MoveL RelTool (p1,30.000000,14.000000,15.535866,\Rx:=0.000000,\Ry:=-4.232438),vel1,zoneval,Extruder\WObj:=Workobject_1;
MoveL RelTool (p1,32.500000,14.000000,16.262071,\Rx:=0.000000,\Ry:=-3.021941),vel1,zoneval,Extruder\WObj:=Workobject_1;
MoveL RelTool (p1,35.000000,14.000000,16.795693,\Rx:=0.000000,\Ry:=-2.300490),vel1,zoneval,Extruder\WObj:=Workobject_1;
MoveL RelTool (p1,37.500000,14.000000,17.167850,\Rx:=0.000000,\Ry:=-1.460854),vel1,zoneval,Extruder\WObj:=Workobject_1;
MoveL RelTool (p1,40.000000,14.000000,17.403542,\Rx:=0.000000,\Ry:=-0.710383),vel1,zoneval,Extruder\WObj:=Workobject_1;
MoveL RelTool (p1,42.500000,14.000000,17.492358,\Rx:=0.000000,\Ry:=0.009614),vel1,zoneval,Extruder\WObj:=Workobject_1;
MoveL RelTool (p1,45.000000,14.000000,17.445886,\Rx:=0.000000,\Ry:=0.497915),vel1,zoneval,Extruder\WObj:=Workobject_1;
MoveL RelTool (p1,47.500000,14.000000,17.268613,\Rx:=0.000000,\Ry:=1.477311),vel1,zoneval,Extruder\WObj:=Workobject_1;
MoveL RelTool (p1,50.000000,14.000000,16.934162,\Rx:=0.000000,\Ry:=1.958454),vel1,zoneval,Extruder\WObj:=Workobject_1;
MoveL RelTool (p1,52.500000,14.000000,16.462457,\Rx:=0.000000,\Ry:=3.004009),vel1,zoneval,Extruder\WObj:=Workobject_1;
MoveL RelTool (p1,55.000000,14.000000,15.799199,\Rx:=0.000000,\Ry:=3.621934),vel1,zoneval,Extruder\WObj:=Workobject_1;
MoveL RelTool (p1,57.500000,14.000000,14.938044,\Rx:=0.000000,\Ry:=4.715755),vel1,zoneval,Extruder\WObj:=Workobject_1;
MoveL RelTool (p1,60.000000,14.000000,13.810971,\Rx:=0.000000,\Ry:=6.022619),vel1,zoneval,Extruder\WObj:=Workobject_1;
MoveL RelTool (p1,62.500000,14.000000,12.303856,\Rx:=0.000000,\Ry:=8.132481),vel1,zoneval,Extruder\WObj:=Workobject_1;
MoveL RelTool (p1,65.000000,14.000000,10.061417,\Rx:=0.000000,\Ry:=11.488801),vel1,zoneval,Extruder\WObj:=Workobject_1;
MoveL RelTool (p1,67.500000,14.000000,7.780757,\Rx:=0.000000,\Ry:=3.821551),vel1,zoneval,Extruder\WObj:=Workobject_1;
MoveL RelTool (p1,70.000000,14.000000,7.500000,\Rx:=0.000000,\Ry:=-0.000000),vel1,zoneval,Extruder\WObj:=Workobject_1;
MoveL RelTool (p1,72.500000,14.000000,7.500000,\Rx:=0.000000,\Ry:=-0.000000),vel1,zoneval,Extruder\WObj:=Workobject_1;
MoveL RelTool (p1,75.000000,14.000000,7.500000,\Rx:=0.000000,\Ry:=-0.000000),vel1,zoneval,Extruder\WObj:=Workobject_1;
MoveL RelTool (p1,77.500000,14.000000,7.500000,\Rx:=0.000000,\Ry:=-0.000000),vel1,zoneval,Extruder\WObj:=Workobject_1;
MoveL RelTool (p1,80.000000,14.000000,7.500000,\Rx:=0.000000,\Ry:=-0.000000),vel1,zoneval,Extruder\WObj:=Workobject_1;
MoveL RelTool (p1,82.500000,14.000000,7.500000,\Rx:=0.000000,\Ry:=-0.000000),vel1,zoneval,Extruder\WObj:=Workobject_1;
MoveL RelTool (p1,80.500000,14.500000,7.500000,\Rx:=0.000000,\Ry:=0.000000),vel1,zoneval,Extruder\WObj:=Workobject_1;
MoveL RelTool (p1,78.000000,14.500000,7.500000,\Rx:=0.000000,\Ry:=0.000000),vel1,zoneval,Extruder\WObj:=Workobject_1;
MoveL RelTool (p1,75.500000,14.500000,7.500000,\Rx:=0.000000,\Ry:=0.000000),vel1,zoneval,Extruder\WObj:=Workobject_1;
MoveL RelTool (p1,73.000000,14.500000,7.500000,\Rx:=0.000000,\Ry:=0.000000),vel1,zoneval,Extruder\WObj:=Workobject_1;
MoveL RelTool (p1,70.500000,14.500000,7.500000,\Rx:=0.000000,\Ry:=0.000000),vel1,zoneval,Extruder\WObj:=Workobject_1;
MoveL RelTool (p1,68.000000,14.500000,7.626010,\Rx:=0.000000,\Ry:=3.821551),vel1,zoneval,Extruder\WObj:=Workobject_1;
MoveL RelTool (p1,65.500000,14.500000,9.428317,\Rx:=0.000000,\Ry:=11.485360),vel1,zoneval,Extruder\WObj:=Workobject_1;
MoveL RelTool (p1,63.000000,14.500000,11.932892,\Rx:=0.000000,\Ry:=8.132481),vel1,zoneval,Extruder\WObj:=Workobject_1;
MoveL RelTool (p1,60.500000,14.500000,13.554932,\Rx:=0.000000,\Ry:=6.053141),vel1,zoneval,Extruder\WObj:=Workobject_1;
MoveL RelTool (p1,58.000000,14.500000,14.744603,\Rx:=0.000000,\Ry:=4.711369),vel1,zoneval,Extruder\WObj:=Workobject_1;
MoveL RelTool (p1,55.500000,14.500000,15.652731,\Rx:=0.000000,\Ry:=3.666878),vel1,zoneval,Extruder\WObj:=Workobject_1;
MoveL RelTool (p1,53.000000,14.500000,16.342269,\Rx:=0.000000,\Ry:=3.014175),vel1,zoneval,Extruder\WObj:=Workobject_1;
MoveL RelTool (p1,50.500000,14.500000,16.857119,\Rx:=0.000000,\Ry:=1.968139),vel1,zoneval,Extruder\WObj:=Workobject_1;
MoveL RelTool (p1,48.000000,14.500000,17.210020,\Rx:=0.000000,\Ry:=1.477311),vel1,zoneval,Extruder\WObj:=Workobject_1;
MoveL RelTool (p1,45.500000,14.500000,17.426141,\Rx:=0.000000,\Ry:=0.497915),vel1,zoneval,Extruder\WObj:=Workobject_1;
MoveL RelTool (p1,43.000000,14.500000,17.491866,\Rx:=0.000000,\Ry:=0.009614),vel1,zoneval,Extruder\WObj:=Workobject_1;
MoveL RelTool (p1,40.500000,14.500000,17.432366,\Rx:=0.000000,\Ry:=-0.740871),vel1,zoneval,Extruder\WObj:=Workobject_1;
MoveL RelTool (p1,38.000000,14.500000,17.226111,\Rx:=0.000000,\Ry:=-1.460854),vel1,zoneval,Extruder\WObj:=Workobject_1;
MoveL RelTool (p1,35.500000,14.500000,16.886724,\Rx:=0.000000,\Ry:=-2.257683),vel1,zoneval,Extruder\WObj:=Workobject_1;
MoveL RelTool (p1,33.000000,14.500000,16.382907,\Rx:=0.000000,\Ry:=-3.021941),vel1,zoneval,Extruder\WObj:=Workobject_1;
MoveL RelTool (p1,30.500000,14.500000,15.708835,\Rx:=0.000000,\Ry:=-4.213102),vel1,zoneval,Extruder\WObj:=Workobject_1;
MoveL RelTool (p1,28.000000,14.500000,14.810880,\Rx:=0.000000,\Ry:=-5.088446),vel1,zoneval,Extruder\WObj:=Workobject_1;
MoveL RelTool (p1,25.500000,14.500000,13.645137,\Rx:=0.000000,\Ry:=-6.516459),vel1,zoneval,Extruder\WObj:=Workobject_1;
MoveL RelTool (p1,23.000000,14.500000,12.058948,\Rx:=0.000000,\Ry:=-8.297239),vel1,zoneval,Extruder\WObj:=Workobject_1;
MoveL RelTool (p1,20.500000,14.500000,9.662581,\Rx:=0.000000,\Ry:=-11.719870),vel1,zoneval,Extruder\WObj:=Workobject_1;
MoveL RelTool (p1,18.000000,14.500000,7.667393,\Rx:=0.000000,\Ry:=-2.952187),vel1,zoneval,Extruder\WObj:=Workobject_1;
MoveL RelTool (p1,15.500000,14.500000,7.500000,\Rx:=0.000000,\Ry:=0.000000),vel1,zoneval,Extruder\WObj:=Workobject_1;
MoveL RelTool (p1,13.000000,14.500000,7.500000,\Rx:=0.000000,\Ry:=0.000000),vel1,zoneval,Extruder\WObj:=Workobject_1;
MoveL RelTool (p1,10.500000,14.500000,7.500000,\Rx:=0.000000,\Ry:=0.000000),vel1,zoneval,Extruder\WObj:=Workobject_1;
MoveL RelTool (p1,8.000000,14.500000,7.500000,\Rx:=0.000000,\Ry:=0.000000),vel1,zoneval,Extruder\WObj:=Workobject_1;
MoveL RelTool (p1,5.500000,14.500000,7.500000,\Rx:=0.000000,\Ry:=0.000000),vel1,zoneval,Extruder\WObj:=Workobject_1;
MoveL RelTool (p1,3.000000,14.500000,7.500000,\Rx:=0.000000,\Ry:=0.000000),vel1,zoneval,Extruder\WObj:=Workobject_1;
MoveL RelTool (p1,5.000000,15.000000,7.500000,\Rx:=0.000000,\Ry:=-0.000000),vel1,zoneval,Extruder\WObj:=Workobject_1;
MoveL RelTool (p1,7.500000,15.000000,7.500000,\Rx:=0.000000,\Ry:=-0.000000),vel1,zoneval,Extruder\WObj:=Workobject_1;
MoveL RelTool (p1,10.000000,15.000000,7.500000,\Rx:=0.000000,\Ry:=-0.000000),vel1,zoneval,Extruder\WObj:=Workobject_1;
MoveL RelTool (p1,12.500000,15.000000,7.500000,\Rx:=0.000000,\Ry:=-0.000000),vel1,zoneval,Extruder\WObj:=Workobject_1;
MoveL RelTool (p1,15.000000,15.000000,7.500000,\Rx:=0.000000,\Ry:=-0.000000),vel1,zoneval,Extruder\WObj:=Workobject_1;
MoveL RelTool (p1,17.500000,15.000000,7.549338,\Rx:=0.000000,\Ry:=-2.952187),vel1,zoneval,Extruder\WObj:=Workobject_1;
MoveL RelTool (p1,20.000000,15.000000,9.005299,\Rx:=0.000000,\Ry:=-11.718071),vel1,zoneval,Extruder\WObj:=Workobject_1;
MoveL RelTool (p1,22.500000,15.000000,11.677302,\Rx:=0.000000,\Ry:=-8.297239),vel1,zoneval,Extruder\WObj:=Workobject_1;
MoveL RelTool (p1,25.000000,15.000000,13.364411,\Rx:=0.000000,\Ry:=-6.507557),vel1,zoneval,Extruder\WObj:=Workobject_1;
MoveL RelTool (p1,27.500000,15.000000,14.600606,\Rx:=0.000000,\Ry:=-5.061360),vel1,zoneval,Extruder\WObj:=Workobject_1;
MoveL RelTool (p1,30.000000,15.000000,15.538278,\Rx:=0.000000,\Ry:=-4.191749),vel1,zoneval,Extruder\WObj:=Workobject_1;
MoveL RelTool (p1,32.500000,15.000000,16.261840,\Rx:=0.000000,\Ry:=-3.021941),vel1,zoneval,Extruder\WObj:=Workobject_1;
MoveL RelTool (p1,35.000000,15.000000,16.798556,\Rx:=0.000000,\Ry:=-2.214824),vel1,zoneval,Extruder\WObj:=Workobject_1;
MoveL RelTool (p1,37.500000,15.000000,17.169131,\Rx:=0.000000,\Ry:=-1.460854),vel1,zoneval,Extruder\WObj:=Workobject_1;
MoveL RelTool (p1,40.000000,15.000000,17.402936,\Rx:=0.000000,\Ry:=-0.761113),vel1,zoneval,Extruder\WObj:=Workobject_1;
MoveL RelTool (p1,42.500000,15.000000,17.492129,\Rx:=0.000000,\Ry:=0.009614),vel1,zoneval,Extruder\WObj:=Workobject_1;
MoveL RelTool (p1,45.000000,15.000000,17.445523,\Rx:=0.000000,\Ry:=0.497915),vel1,zoneval,Extruder\WObj:=Workobject_1;
MoveL RelTool (p1,47.500000,15.000000,17.267978,\Rx:=0.000000,\Ry:=1.477311),vel1,zoneval,Extruder\WObj:=Workobject_1;
MoveL RelTool (p1,50.000000,15.000000,16.935897,\Rx:=0.000000,\Ry:=1.976483),vel1,zoneval,Extruder\WObj:=Workobject_1;
MoveL RelTool (p1,52.500000,15.000000,16.462915,\Rx:=0.000000,\Ry:=3.014175),vel1,zoneval,Extruder\WObj:=Workobject_1;
MoveL RelTool (p1,55.000000,15.000000,15.802495,\Rx:=0.000000,\Ry:=3.711728),vel1,zoneval,Extruder\WObj:=Workobject_1;
MoveL RelTool (p1,57.500000,15.000000,14.939061,\Rx:=0.000000,\Ry:=4.706981),vel1,zoneval,Extruder\WObj:=Workobject_1;
MoveL RelTool (p1,60.000000,15.000000,13.813687,\Rx:=0.000000,\Ry:=6.083587),vel1,zoneval,Extruder\WObj:=Workobject_1;
MoveL RelTool (p1,62.500000,15.000000,12.304491,\Rx:=0.000000,\Ry:=8.132481),vel1,zoneval,Extruder\WObj:=Workobject_1;
MoveL RelTool (p1,65.000000,15.000000,10.060714,\Rx:=0.000000,\Ry:=11.481917),vel1,zoneval,Extruder\WObj:=Workobject_1;
MoveL RelTool (p1,67.500000,15.000000,7.780757,\Rx:=0.000000,\Ry:=3.821551),vel1,zoneval,Extruder\WObj:=Workobject_1;
MoveL RelTool (p1,70.000000,15.000000,7.500000,\Rx:=0.000000,\Ry:=-0.000000),vel1,zoneval,Extruder\WObj:=Workobject_1;
MoveL RelTool (p1,72.500000,15.000000,7.500000,\Rx:=0.000000,\Ry:=-0.000000),vel1,zoneval,Extruder\WObj:=Workobject_1;
MoveL RelTool (p1,75.000000,15.000000,7.500000,\Rx:=0.000000,\Ry:=-0.000000),vel1,zoneval,Extruder\WObj:=Workobject_1;
MoveL RelTool (p1,77.500000,15.000000,7.500000,\Rx:=0.000000,\Ry:=-0.000000),vel1,zoneval,Extruder\WObj:=Workobject_1;
MoveL RelTool (p1,80.000000,15.000000,7.500000,\Rx:=0.000000,\Ry:=-0.000000),vel1,zoneval,Extruder\WObj:=Workobject_1;
MoveL RelTool (p1,82.500000,15.000000,7.500000,\Rx:=0.000000,\Ry:=-0.000000),vel1,zoneval,Extruder\WObj:=Workobject_1;
MoveL RelTool (p1,80.500000,15.500000,7.500000,\Rx:=0.000000,\Ry:=0.000000),vel1,zoneval,Extruder\WObj:=Workobject_1;
MoveL RelTool (p1,78.000000,15.500000,7.500000,\Rx:=0.000000,\Ry:=0.000000),vel1,zoneval,Extruder\WObj:=Workobject_1;
MoveL RelTool (p1,75.500000,15.500000,7.500000,\Rx:=0.000000,\Ry:=0.000000),vel1,zoneval,Extruder\WObj:=Workobject_1;
MoveL RelTool (p1,73.000000,15.500000,7.500000,\Rx:=0.000000,\Ry:=0.000000),vel1,zoneval,Extruder\WObj:=Workobject_1;
MoveL RelTool (p1,70.500000,15.500000,7.500000,\Rx:=0.000000,\Ry:=0.000000),vel1,zoneval,Extruder\WObj:=Workobject_1;
MoveL RelTool (p1,68.000000,15.500000,7.626010,\Rx:=0.000000,\Ry:=3.821551),vel1,zoneval,Extruder\WObj:=Workobject_1;
MoveL RelTool (p1,65.500000,15.500000,9.428317,\Rx:=0.000000,\Ry:=11.478472),vel1,zoneval,Extruder\WObj:=Workobject_1;
MoveL RelTool (p1,63.000000,15.500000,11.933528,\Rx:=0.000000,\Ry:=8.132481),vel1,zoneval,Extruder\WObj:=Workobject_1;
MoveL RelTool (p1,60.500000,15.500000,13.554619,\Rx:=0.000000,\Ry:=6.113959),vel1,zoneval,Extruder\WObj:=Workobject_1;
MoveL RelTool (p1,58.000000,15.500000,14.746017,\Rx:=0.000000,\Ry:=4.702592),vel1,zoneval,Extruder\WObj:=Workobject_1;
MoveL RelTool (p1,55.500000,15.500000,15.652192,\Rx:=0.000000,\Ry:=3.756483),vel1,zoneval,Extruder\WObj:=Workobject_1;
MoveL RelTool (p1,53.000000,15.500000,16.342305,\Rx:=0.000000,\Ry:=3.014175),vel1,zoneval,Extruder\WObj:=Workobject_1;
MoveL RelTool (p1,50.500000,15.500000,16.858518,\Rx:=0.000000,\Ry:=1.976483),vel1,zoneval,Extruder\WObj:=Workobject_1;
MoveL RelTool (p1,48.000000,15.500000,17.209385,\Rx:=0.000000,\Ry:=1.477311),vel1,zoneval,Extruder\WObj:=Workobject_1;
MoveL RelTool (p1,45.500000,15.500000,17.425779,\Rx:=0.000000,\Ry:=0.497915),vel1,zoneval,Extruder\WObj:=Workobject_1;
MoveL RelTool (p1,43.000000,15.500000,17.491637,\Rx:=0.000000,\Ry:=0.009614),vel1,zoneval,Extruder\WObj:=Workobject_1;
MoveL RelTool (p1,40.500000,15.500000,17.433003,\Rx:=0.000000,\Ry:=-0.772436),vel1,zoneval,Extruder\WObj:=Workobject_1;
MoveL RelTool (p1,38.000000,15.500000,17.227393,\Rx:=0.000000,\Ry:=-1.460854),vel1,zoneval,Extruder\WObj:=Workobject_1;
MoveL RelTool (p1,35.500000,15.500000,16.886115,\Rx:=0.000000,\Ry:=-2.171914),vel1,zoneval,Extruder\WObj:=Workobject_1;
MoveL RelTool (p1,33.000000,15.500000,16.382676,\Rx:=0.000000,\Ry:=-3.021941),vel1,zoneval,Extruder\WObj:=Workobject_1;
MoveL RelTool (p1,30.500000,15.500000,15.708951,\Rx:=0.000000,\Ry:=-4.160740),vel1,zoneval,Extruder\WObj:=Workobject_1;
MoveL RelTool (p1,28.000000,15.500000,14.810202,\Rx:=0.000000,\Ry:=-5.034225),vel1,zoneval,Extruder\WObj:=Workobject_1;
MoveL RelTool (p1,25.500000,15.500000,13.644491,\Rx:=0.000000,\Ry:=-6.498647),vel1,zoneval,Extruder\WObj:=Workobject_1;
MoveL RelTool (p1,23.000000,15.500000,12.058489,\Rx:=0.000000,\Ry:=-8.297239),vel1,zoneval,Extruder\WObj:=Workobject_1;
MoveL RelTool (p1,20.500000,15.500000,9.662195,\Rx:=0.000000,\Ry:=-11.716271),vel1,zoneval,Extruder\WObj:=Workobject_1;
MoveL RelTool (p1,18.000000,15.500000,7.667393,\Rx:=0.000000,\Ry:=-2.952187),vel1,zoneval,Extruder\WObj:=Workobject_1;
MoveL RelTool (p1,15.500000,15.500000,7.500000,\Rx:=0.000000,\Ry:=0.000000),vel1,zoneval,Extruder\WObj:=Workobject_1;
MoveL RelTool (p1,13.000000,15.500000,7.500000,\Rx:=0.000000,\Ry:=0.000000),vel1,zoneval,Extruder\WObj:=Workobject_1;
MoveL RelTool (p1,10.500000,15.500000,7.500000,\Rx:=0.000000,\Ry:=0.000000),vel1,zoneval,Extruder\WObj:=Workobject_1;
MoveL RelTool (p1,8.000000,15.500000,7.500000,\Rx:=0.000000,\Ry:=0.000000),vel1,zoneval,Extruder\WObj:=Workobject_1;
MoveL RelTool (p1,5.500000,15.500000,7.500000,\Rx:=0.000000,\Ry:=0.000000),vel1,zoneval,Extruder\WObj:=Workobject_1;
MoveL RelTool (p1,3.000000,15.500000,7.500000,\Rx:=0.000000,\Ry:=0.000000),vel1,zoneval,Extruder\WObj:=Workobject_1;
MoveL RelTool (p1,5.000000,16.000000,7.500000,\Rx:=0.000000,\Ry:=-0.000000),vel1,zoneval,Extruder\WObj:=Workobject_1;
MoveL RelTool (p1,7.500000,16.000000,7.500000,\Rx:=0.000000,\Ry:=-0.000000),vel1,zoneval,Extruder\WObj:=Workobject_1;
MoveL RelTool (p1,10.000000,16.000000,7.500000,\Rx:=0.000000,\Ry:=-0.000000),vel1,zoneval,Extruder\WObj:=Workobject_1;
MoveL RelTool (p1,12.500000,16.000000,7.500000,\Rx:=0.000000,\Ry:=-0.000000),vel1,zoneval,Extruder\WObj:=Workobject_1;
MoveL RelTool (p1,15.000000,16.000000,7.500000,\Rx:=0.000000,\Ry:=-0.000000),vel1,zoneval,Extruder\WObj:=Workobject_1;
MoveL RelTool (p1,17.500000,16.000000,7.549338,\Rx:=0.000000,\Ry:=-2.952187),vel1,zoneval,Extruder\WObj:=Workobject_1;
MoveL RelTool (p1,20.000000,16.000000,9.005299,\Rx:=0.000000,\Ry:=-11.714470),vel1,zoneval,Extruder\WObj:=Workobject_1;
MoveL RelTool (p1,22.500000,16.000000,11.676843,\Rx:=0.000000,\Ry:=-8.297239),vel1,zoneval,Extruder\WObj:=Workobject_1;
MoveL RelTool (p1,25.000000,16.000000,13.364684,\Rx:=0.000000,\Ry:=-6.489730),vel1,zoneval,Extruder\WObj:=Workobject_1;
MoveL RelTool (p1,27.500000,16.000000,14.602432,\Rx:=0.000000,\Ry:=-5.007042),vel1,zoneval,Extruder\WObj:=Workobject_1;
MoveL RelTool (p1,30.000000,16.000000,15.540690,\Rx:=0.000000,\Ry:=-4.129681),vel1,zoneval,Extruder\WObj:=Workobject_1;
MoveL RelTool (p1,32.500000,16.000000,16.261609,\Rx:=0.000000,\Ry:=-3.021941),vel1,zoneval,Extruder\WObj:=Workobject_1;
MoveL RelTool (p1,35.000000,16.000000,16.801419,\Rx:=0.000000,\Ry:=-2.128954),vel1,zoneval,Extruder\WObj:=Workobject_1;
MoveL RelTool (p1,37.500000,16.000000,17.170413,\Rx:=0.000000,\Ry:=-1.460854),vel1,zoneval,Extruder\WObj:=Workobject_1;
MoveL RelTool (p1,40.000000,16.000000,17.402329,\Rx:=0.000000,\Ry:=-0.783758),vel1,zoneval,Extruder\WObj:=Workobject_1;
MoveL RelTool (p1,42.500000,16.000000,17.491899,\Rx:=0.000000,\Ry:=0.009614),vel1,zoneval,Extruder\WObj:=Workobject_1;
MoveL RelTool (p1,45.000000,16.000000,17.445161,\Rx:=0.000000,\Ry:=0.497915),vel1,zoneval,Extruder\WObj:=Workobject_1;
MoveL RelTool (p1,47.500000,16.000000,17.267343,\Rx:=0.000000,\Ry:=1.477311),vel1,zoneval,Extruder\WObj:=Workobject_1;
MoveL RelTool (p1,50.000000,16.000000,16.937631,\Rx:=0.000000,\Ry:=1.976483),vel1,zoneval,Extruder\WObj:=Workobject_1;
MoveL RelTool (p1,52.500000,16.000000,16.462951,\Rx:=0.000000,\Ry:=3.014175),vel1,zoneval,Extruder\WObj:=Workobject_1;
MoveL RelTool (p1,55.000000,16.000000,15.805792,\Rx:=0.000000,\Ry:=3.801143),vel1,zoneval,Extruder\WObj:=Workobject_1;
MoveL RelTool (p1,57.500000,16.000000,14.940078,\Rx:=0.000000,\Ry:=4.700199),vel1,zoneval,Extruder\WObj:=Workobject_1;
MoveL RelTool (p1,60.000000,16.000000,13.816402,\Rx:=0.000000,\Ry:=6.144255),vel1,zoneval,Extruder\WObj:=Workobject_1;
MoveL RelTool (p1,62.500000,16.000000,12.305126,\Rx:=0.000000,\Ry:=8.132481),vel1,zoneval,Extruder\WObj:=Workobject_1;
MoveL RelTool (p1,65.000000,16.000000,10.060011,\Rx:=0.000000,\Ry:=11.475024),vel1,zoneval,Extruder\WObj:=Workobject_1;
MoveL RelTool (p1,67.500000,16.000000,7.780757,\Rx:=0.000000,\Ry:=3.821551),vel1,zoneval,Extruder\WObj:=Workobject_1;
MoveL RelTool (p1,70.000000,16.000000,7.500000,\Rx:=0.000000,\Ry:=-0.000000),vel1,zoneval,Extruder\WObj:=Workobject_1;
MoveL RelTool (p1,72.500000,16.000000,7.500000,\Rx:=0.000000,\Ry:=-0.000000),vel1,zoneval,Extruder\WObj:=Workobject_1;
MoveL RelTool (p1,75.000000,16.000000,7.500000,\Rx:=0.000000,\Ry:=-0.000000),vel1,zoneval,Extruder\WObj:=Workobject_1;
MoveL RelTool (p1,77.500000,16.000000,7.500000,\Rx:=0.000000,\Ry:=-0.000000),vel1,zoneval,Extruder\WObj:=Workobject_1;
MoveL RelTool (p1,80.000000,16.000000,7.500000,\Rx:=0.000000,\Ry:=-0.000000),vel1,zoneval,Extruder\WObj:=Workobject_1;
MoveL RelTool (p1,82.500000,16.000000,7.500000,\Rx:=0.000000,\Ry:=-0.000000),vel1,zoneval,Extruder\WObj:=Workobject_1;




MoveL RelTool (p1,82.500000,16.000000,70.00000,\Rx:=0.000000,\Ry:=-0.000000),vel1,zoneval,Extruder\WObj:=Workobject_1;


MoveL RelTool (p1,3.000000,3.000000,70.000000,\Rx:=0.000000,\Ry:=0.000000),vel1,z0,Extruder\WObj:=Workobject_1;

MoveL RelTool (p1,3.000000,3.000000,8.000000,\Rx:=0.000000,\Ry:=0.000000),vel1,z0,Extruder\WObj:=Workobject_1;
MoveL RelTool (p1,16.889791,3.000000,8.000000,\Rx:=0.000000,\Ry:=0.000000),vel1,z0,Extruder\WObj:=Workobject_1;
MoveL RelTool (p1,17.452093,3.000000,8.045464,\Rx:=0.000000,\Ry:=0.000000),vel1,z0,Extruder\WObj:=Workobject_1;
MoveL RelTool (p1,17.999786,3.000000,8.180676,\Rx:=0.000000,\Ry:=0.000000),vel1,z0,Extruder\WObj:=Workobject_1;
MoveL RelTool (p1,18.518642,3.000000,8.402122,\Rx:=0.000000,\Ry:=0.000000),vel1,z0,Extruder\WObj:=Workobject_1;
MoveL RelTool (p1,18.995180,3.000000,8.704050,\Rx:=0.000000,\Ry:=0.000000),vel1,z0,Extruder\WObj:=Workobject_1;
MoveL RelTool (p1,19.417023,3.000000,9.078616,\Rx:=0.000000,\Ry:=0.000000),vel1,z0,Extruder\WObj:=Workobject_1;
MoveL RelTool (p1,19.773207,3.000000,9.516088,\Rx:=0.000000,\Ry:=0.000000),vel1,z0,Extruder\WObj:=Workobject_1;
MoveL RelTool (p1,20.250246,3.000000,10.153003,\Rx:=0.000000,\Ry:=0.000000),vel1,z0,Extruder\WObj:=Workobject_1;
MoveL RelTool (p1,21.342972,3.000000,11.327476,\Rx:=0.000000,\Ry:=0.000000),vel1,z0,Extruder\WObj:=Workobject_1;
MoveL RelTool (p1,22.725681,3.000000,12.487259,\Rx:=0.000000,\Ry:=0.000000),vel1,z0,Extruder\WObj:=Workobject_1;
MoveL RelTool (p1,24.403374,3.000000,13.604031,\Rx:=0.000000,\Ry:=0.000000),vel1,z0,Extruder\WObj:=Workobject_1;
MoveL RelTool (p1,26.408426,3.000000,14.665359,\Rx:=0.000000,\Ry:=0.000000),vel1,z0,Extruder\WObj:=Workobject_1;
MoveL RelTool (p1,28.691647,3.000000,15.620553,\Rx:=0.000000,\Ry:=0.000000),vel1,z0,Extruder\WObj:=Workobject_1;
MoveL RelTool (p1,31.195286,3.000000,16.437975,\Rx:=0.000000,\Ry:=0.000000),vel1,z0,Extruder\WObj:=Workobject_1;
MoveL RelTool (p1,33.926628,3.000000,17.106159,\Rx:=0.000000,\Ry:=0.000000),vel1,z0,Extruder\WObj:=Workobject_1;
MoveL RelTool (p1,36.846878,3.000000,17.599693,\Rx:=0.000000,\Ry:=0.000000),vel1,z0,Extruder\WObj:=Workobject_1;
MoveL RelTool (p1,39.856747,3.000000,17.899025,\Rx:=0.000000,\Ry:=0.000000),vel1,z0,Extruder\WObj:=Workobject_1;
MoveL RelTool (p1,42.916187,3.000000,18.000000,\Rx:=0.000000,\Ry:=0.000000),vel1,z0,Extruder\WObj:=Workobject_1;
MoveL RelTool (p1,45.700897,3.000000,17.916361,\Rx:=0.000000,\Ry:=0.000000),vel1,z0,Extruder\WObj:=Workobject_1;
MoveL RelTool (p1,48.678219,3.000000,17.639635,\Rx:=0.000000,\Ry:=0.000000),vel1,z0,Extruder\WObj:=Workobject_1;
MoveL RelTool (p1,51.519215,3.000000,17.183882,\Rx:=0.000000,\Ry:=0.000000),vel1,z0,Extruder\WObj:=Workobject_1;
MoveL RelTool (p1,54.218540,3.000000,16.554611,\Rx:=0.000000,\Ry:=0.000000),vel1,z0,Extruder\WObj:=Workobject_1;
MoveL RelTool (p1,56.711525,3.000000,15.776219,\Rx:=0.000000,\Ry:=0.000000),vel1,z0,Extruder\WObj:=Workobject_1;
MoveL RelTool (p1,58.923611,3.000000,14.894774,\Rx:=0.000000,\Ry:=0.000000),vel1,z0,Extruder\WObj:=Workobject_1;
MoveL RelTool (p1,60.880539,3.000000,13.919682,\Rx:=0.000000,\Ry:=0.000000),vel1,z0,Extruder\WObj:=Workobject_1;
MoveL RelTool (p1,62.570816,3.000000,12.872232,\Rx:=0.000000,\Ry:=0.000000),vel1,z0,Extruder\WObj:=Workobject_1;
MoveL RelTool (p1,63.995117,3.000000,11.774377,\Rx:=0.000000,\Ry:=0.000000),vel1,z0,Extruder\WObj:=Workobject_1;
MoveL RelTool (p1,65.148392,3.000000,10.656720,\Rx:=0.000000,\Ry:=0.000000),vel1,z0,Extruder\WObj:=Workobject_1;
MoveL RelTool (p1,66.059166,3.000000,9.516088,\Rx:=0.000000,\Ry:=0.000000),vel1,z0,Extruder\WObj:=Workobject_1;
MoveL RelTool (p1,66.415344,3.000000,9.078616,\Rx:=0.000000,\Ry:=0.000000),vel1,z0,Extruder\WObj:=Workobject_1;
MoveL RelTool (p1,66.837189,3.000000,8.704050,\Rx:=0.000000,\Ry:=0.000000),vel1,z0,Extruder\WObj:=Workobject_1;
MoveL RelTool (p1,67.313728,3.000000,8.402122,\Rx:=0.000000,\Ry:=0.000000),vel1,z0,Extruder\WObj:=Workobject_1;
MoveL RelTool (p1,67.832588,3.000000,8.180676,\Rx:=0.000000,\Ry:=0.000000),vel1,z0,Extruder\WObj:=Workobject_1;
MoveL RelTool (p1,68.380280,3.000000,8.045464,\Rx:=0.000000,\Ry:=0.000000),vel1,z0,Extruder\WObj:=Workobject_1;
MoveL RelTool (p1,68.942581,3.000000,8.000000,\Rx:=0.000000,\Ry:=0.000000),vel1,z0,Extruder\WObj:=Workobject_1;
MoveL RelTool (p1,82.832375,3.000000,8.000000,\Rx:=0.000000,\Ry:=0.000000),vel1,z0,Extruder\WObj:=Workobject_1;
MoveL RelTool (p1,82.832375,16.000000,8.000000,\Rx:=0.000000,\Ry:=0.000000),vel1,z0,Extruder\WObj:=Workobject_1;
MoveL RelTool (p1,68.942581,16.000000,8.000000,\Rx:=0.000000,\Ry:=0.000000),vel1,z0,Extruder\WObj:=Workobject_1;
MoveL RelTool (p1,68.380280,16.000000,8.045464,\Rx:=0.000000,\Ry:=0.000000),vel1,z0,Extruder\WObj:=Workobject_1;
MoveL RelTool (p1,67.832588,16.000000,8.180676,\Rx:=0.000000,\Ry:=0.000000),vel1,z0,Extruder\WObj:=Workobject_1;
MoveL RelTool (p1,67.313728,16.000000,8.402122,\Rx:=0.000000,\Ry:=0.000000),vel1,z0,Extruder\WObj:=Workobject_1;
MoveL RelTool (p1,66.837189,16.000000,8.704050,\Rx:=0.000000,\Ry:=0.000000),vel1,z0,Extruder\WObj:=Workobject_1;
MoveL RelTool (p1,66.415344,16.000000,9.078616,\Rx:=0.000000,\Ry:=0.000000),vel1,z0,Extruder\WObj:=Workobject_1;
MoveL RelTool (p1,66.059166,16.000000,9.516088,\Rx:=0.000000,\Ry:=0.000000),vel1,z0,Extruder\WObj:=Workobject_1;
MoveL RelTool (p1,65.564453,16.000000,10.174875,\Rx:=0.000000,\Ry:=0.000000),vel1,z0,Extruder\WObj:=Workobject_1;
MoveL RelTool (p1,65.143768,16.000000,10.652657,\Rx:=0.000000,\Ry:=0.000000),vel1,z0,Extruder\WObj:=Workobject_1;
MoveL RelTool (p1,64.991638,16.000000,10.825450,\Rx:=0.000000,\Ry:=0.000000),vel1,z0,Extruder\WObj:=Workobject_1;
MoveL RelTool (p1,64.322777,16.000000,11.482923,\Rx:=0.000000,\Ry:=0.000000),vel1,z0,Extruder\WObj:=Workobject_1;
MoveL RelTool (p1,63.989872,16.000000,11.768258,\Rx:=0.000000,\Ry:=0.000000),vel1,z0,Extruder\WObj:=Workobject_1;
MoveL RelTool (p1,63.561058,16.000000,12.135797,\Rx:=0.000000,\Ry:=0.000000),vel1,z0,Extruder\WObj:=Workobject_1;
MoveL RelTool (p1,62.719486,16.000000,12.768417,\Rx:=0.000000,\Ry:=0.000000),vel1,z0,Extruder\WObj:=Workobject_1;
MoveL RelTool (p1,62.568321,16.000000,12.868458,\Rx:=0.000000,\Ry:=0.000000),vel1,z0,Extruder\WObj:=Workobject_1;
MoveL RelTool (p1,61.766850,16.000000,13.398852,\Rx:=0.000000,\Ry:=0.000000),vel1,z0,Extruder\WObj:=Workobject_1;
MoveL RelTool (p1,60.878704,16.000000,13.916541,\Rx:=0.000000,\Ry:=0.000000),vel1,z0,Extruder\WObj:=Workobject_1;
MoveL RelTool (p1,60.738800,16.000000,13.998090,\Rx:=0.000000,\Ry:=0.000000),vel1,z0,Extruder\WObj:=Workobject_1;
MoveL RelTool (p1,59.623398,16.000000,14.570664,\Rx:=0.000000,\Ry:=0.000000),vel1,z0,Extruder\WObj:=Workobject_1;
MoveL RelTool (p1,58.920467,16.000000,14.887815,\Rx:=0.000000,\Ry:=0.000000),vel1,z0,Extruder\WObj:=Workobject_1;
MoveL RelTool (p1,58.413136,16.000000,15.116714,\Rx:=0.000000,\Ry:=0.000000),vel1,z0,Extruder\WObj:=Workobject_1;
MoveL RelTool (p1,57.100113,16.000000,15.635588,\Rx:=0.000000,\Ry:=0.000000),vel1,z0,Extruder\WObj:=Workobject_1;
MoveL RelTool (p1,56.709370,16.000000,15.769944,\Rx:=0.000000,\Ry:=0.000000),vel1,z0,Extruder\WObj:=Workobject_1;
MoveL RelTool (p1,55.682240,16.000000,16.123117,\Rx:=0.000000,\Ry:=0.000000),vel1,z0,Extruder\WObj:=Workobject_1;
MoveL RelTool (p1,54.218712,16.000000,16.555187,\Rx:=0.000000,\Ry:=0.000000),vel1,z0,Extruder\WObj:=Workobject_1;
MoveL RelTool (p1,54.214844,16.000000,16.556330,\Rx:=0.000000,\Ry:=0.000000),vel1,z0,Extruder\WObj:=Workobject_1;
MoveL RelTool (p1,52.687428,16.000000,16.937145,\Rx:=0.000000,\Ry:=0.000000),vel1,z0,Extruder\WObj:=Workobject_1;
MoveL RelTool (p1,51.517960,16.000000,17.177769,\Rx:=0.000000,\Ry:=0.000000),vel1,z0,Extruder\WObj:=Workobject_1;
MoveL RelTool (p1,51.097290,16.000000,17.264324,\Rx:=0.000000,\Ry:=0.000000),vel1,z0,Extruder\WObj:=Workobject_1;
MoveL RelTool (p1,49.441021,16.000000,17.536478,\Rx:=0.000000,\Ry:=0.000000),vel1,z0,Extruder\WObj:=Workobject_1;
MoveL RelTool (p1,48.677208,16.000000,17.631521,\Rx:=0.000000,\Ry:=0.000000),vel1,z0,Extruder\WObj:=Workobject_1;
MoveL RelTool (p1,47.734676,16.000000,17.748802,\Rx:=0.000000,\Ry:=0.000000),vel1,z0,Extruder\WObj:=Workobject_1;
MoveL RelTool (p1,45.987778,16.000000,17.898254,\Rx:=0.000000,\Ry:=0.000000),vel1,z0,Extruder\WObj:=Workobject_1;
MoveL RelTool (p1,45.700684,16.000000,17.911810,\Rx:=0.000000,\Ry:=0.000000),vel1,z0,Extruder\WObj:=Workobject_1;
MoveL RelTool (p1,44.220581,16.000000,17.981699,\Rx:=0.000000,\Ry:=0.000000),vel1,z0,Extruder\WObj:=Workobject_1;
MoveL RelTool (p1,42.916126,16.000000,17.993467,\Rx:=0.000000,\Ry:=0.000000),vel1,z0,Extruder\WObj:=Workobject_1;
MoveL RelTool (p1,42.450130,16.000000,17.997671,\Rx:=0.000000,\Ry:=0.000000),vel1,z0,Extruder\WObj:=Workobject_1;
MoveL RelTool (p1,40.680767,16.000000,17.946178,\Rx:=0.000000,\Ry:=0.000000),vel1,z0,Extruder\WObj:=Workobject_1;
MoveL RelTool (p1,39.857311,16.000000,17.890665,\Rx:=0.000000,\Ry:=0.000000),vel1,z0,Extruder\WObj:=Workobject_1;
MoveL RelTool (p1,38.917850,16.000000,17.827332,\Rx:=0.000000,\Ry:=0.000000),vel1,z0,Extruder\WObj:=Workobject_1;
MoveL RelTool (p1,37.181221,16.000000,17.643127,\Rx:=0.000000,\Ry:=0.000000),vel1,z0,Extruder\WObj:=Workobject_1;
MoveL RelTool (p1,36.847645,16.000000,17.594460,\Rx:=0.000000,\Ry:=0.000000),vel1,z0,Extruder\WObj:=Workobject_1;
MoveL RelTool (p1,35.475056,16.000000,17.394205,\Rx:=0.000000,\Ry:=0.000000),vel1,z0,Extruder\WObj:=Workobject_1;
MoveL RelTool (p1,33.926945,16.000000,17.104464,\Rx:=0.000000,\Ry:=0.000000),vel1,z0,Extruder\WObj:=Workobject_1;
MoveL RelTool (p1,33.825615,16.000000,17.085497,\Rx:=0.000000,\Ry:=0.000000),vel1,z0,Extruder\WObj:=Workobject_1;
MoveL RelTool (p1,32.239231,16.000000,16.719597,\Rx:=0.000000,\Ry:=0.000000),vel1,z0,Extruder\WObj:=Workobject_1;
MoveL RelTool (p1,31.197088,16.000000,16.431459,\Rx:=0.000000,\Ry:=0.000000),vel1,z0,Extruder\WObj:=Workobject_1;
MoveL RelTool (p1,30.718615,16.000000,16.299169,\Rx:=0.000000,\Ry:=0.000000),vel1,z0,Extruder\WObj:=Workobject_1;
MoveL RelTool (p1,29.260920,16.000000,15.825695,\Rx:=0.000000,\Ry:=0.000000),vel1,z0,Extruder\WObj:=Workobject_1;
MoveL RelTool (p1,28.694523,16.000000,15.612896,\Rx:=0.000000,\Ry:=0.000000),vel1,z0,Extruder\WObj:=Workobject_1;
MoveL RelTool (p1,27.880777,16.000000,15.307163,\Rx:=0.000000,\Ry:=0.000000),vel1,z0,Extruder\WObj:=Workobject_1;
MoveL RelTool (p1,26.594425,16.000000,14.752407,\Rx:=0.000000,\Ry:=0.000000),vel1,z0,Extruder\WObj:=Workobject_1;
MoveL RelTool (p1,26.410309,16.000000,14.661544,\Rx:=0.000000,\Ry:=0.000000),vel1,z0,Extruder\WObj:=Workobject_1;
MoveL RelTool (p1,25.404926,16.000000,14.165370,\Rx:=0.000000,\Ry:=0.000000),vel1,z0,Extruder\WObj:=Workobject_1;
MoveL RelTool (p1,24.404613,16.000000,13.601830,\Rx:=0.000000,\Ry:=0.000000),vel1,z0,Extruder\WObj:=Workobject_1;
MoveL RelTool (p1,24.315626,16.000000,13.551698,\Rx:=0.000000,\Ry:=0.000000),vel1,z0,Extruder\WObj:=Workobject_1;
MoveL RelTool (p1,23.320549,16.000000,12.912832,\Rx:=0.000000,\Ry:=0.000000),vel1,z0,Extruder\WObj:=Workobject_1;
MoveL RelTool (p1,22.730097,16.000000,12.481217,\Rx:=0.000000,\Ry:=0.000000),vel1,z0,Extruder\WObj:=Workobject_1;
MoveL RelTool (p1,22.437567,16.000000,12.267382,\Rx:=0.000000,\Ry:=0.000000),vel1,z0,Extruder\WObj:=Workobject_1;
MoveL RelTool (p1,21.638329,16.000000,11.599616,\Rx:=0.000000,\Ry:=0.000000),vel1,z0,Extruder\WObj:=Workobject_1;
MoveL RelTool (p1,21.348730,16.000000,11.321481,\Rx:=0.000000,\Ry:=0.000000),vel1,z0,Extruder\WObj:=Workobject_1;
MoveL RelTool (p1,20.937675,16.000000,10.926694,\Rx:=0.000000,\Ry:=0.000000),vel1,z0,Extruder\WObj:=Workobject_1;
MoveL RelTool (p1,20.332558,16.000000,10.253466,\Rx:=0.000000,\Ry:=0.000000),vel1,z0,Extruder\WObj:=Workobject_1;
MoveL RelTool (p1,20.253410,16.000000,10.150568,\Rx:=0.000000,\Ry:=0.000000),vel1,z0,Extruder\WObj:=Workobject_1;
MoveL RelTool (p1,19.850492,16.000000,9.626740,\Rx:=0.000000,\Ry:=0.000000),vel1,z0,Extruder\WObj:=Workobject_1;
MoveL RelTool (p1,19.773207,16.000000,9.516088,\Rx:=0.000000,\Ry:=0.000000),vel1,z0,Extruder\WObj:=Workobject_1;
MoveL RelTool (p1,19.417023,16.000000,9.078616,\Rx:=0.000000,\Ry:=0.000000),vel1,z0,Extruder\WObj:=Workobject_1;
MoveL RelTool (p1,18.995180,16.000000,8.704050,\Rx:=0.000000,\Ry:=0.000000),vel1,z0,Extruder\WObj:=Workobject_1;
MoveL RelTool (p1,18.518642,16.000000,8.402122,\Rx:=0.000000,\Ry:=0.000000),vel1,z0,Extruder\WObj:=Workobject_1;
MoveL RelTool (p1,17.999786,16.000000,8.180676,\Rx:=0.000000,\Ry:=0.000000),vel1,z0,Extruder\WObj:=Workobject_1;
MoveL RelTool (p1,17.452093,16.000000,8.045464,\Rx:=0.000000,\Ry:=0.000000),vel1,z0,Extruder\WObj:=Workobject_1;
MoveL RelTool (p1,16.889791,16.000000,8.000000,\Rx:=0.000000,\Ry:=0.000000),vel1,z0,Extruder\WObj:=Workobject_1;
MoveL RelTool (p1,3.000000,16.000000,8.000000,\Rx:=0.000000,\Ry:=0.000000),vel1,z0,Extruder\WObj:=Workobject_1;
MoveL RelTool (p1,3.000000,3.000000,8.000000,\Rx:=0.000000,\Ry:=0.000000),vel1,z0,Extruder\WObj:=Workobject_1;





MoveL RelTool (p1,3.000000,3.000000,8.000000,\Rx:=0.000000,\Ry:=0),vel1,zoneval,Extruder\WObj:=Workobject_1;
MoveL RelTool (p1,5.000000,3.000000,8.000000,\Rx:=0.000000,\Ry:=-0.000000),vel1,zoneval,Extruder\WObj:=Workobject_1;
MoveL RelTool (p1,7.500000,3.000000,8.000000,\Rx:=0.000000,\Ry:=-0.000000),vel1,zoneval,Extruder\WObj:=Workobject_1;
MoveL RelTool (p1,10.000000,3.000000,8.000000,\Rx:=0.000000,\Ry:=-0.000000),vel1,zoneval,Extruder\WObj:=Workobject_1;
MoveL RelTool (p1,12.500000,3.000000,8.000000,\Rx:=0.000000,\Ry:=-0.000000),vel1,zoneval,Extruder\WObj:=Workobject_1;
MoveL RelTool (p1,15.000000,3.000000,8.000000,\Rx:=0.000000,\Ry:=-0.000000),vel1,zoneval,Extruder\WObj:=Workobject_1;
MoveL RelTool (p1,17.500000,3.000000,8.057291,\Rx:=0.000000,\Ry:=-3.082616),vel1,zoneval,Extruder\WObj:=Workobject_1;
MoveL RelTool (p1,20.000000,3.000000,9.818889,\Rx:=0.000000,\Ry:=-11.180880),vel1,zoneval,Extruder\WObj:=Workobject_1;
MoveL RelTool (p1,22.500000,3.000000,12.297963,\Rx:=0.000000,\Ry:=-8.142619),vel1,zoneval,Extruder\WObj:=Workobject_1;
MoveL RelTool (p1,25.000000,3.000000,13.919841,\Rx:=0.000000,\Ry:=-6.198553),vel1,zoneval,Extruder\WObj:=Workobject_1;
MoveL RelTool (p1,27.500000,3.000000,15.122023,\Rx:=0.000000,\Ry:=-5.044928),vel1,zoneval,Extruder\WObj:=Workobject_1;
MoveL RelTool (p1,30.000000,3.000000,16.047722,\Rx:=0.000000,\Ry:=-4.018116),vel1,zoneval,Extruder\WObj:=Workobject_1;
MoveL RelTool (p1,32.500000,3.000000,16.757155,\Rx:=0.000000,\Ry:=-3.054804),vel1,zoneval,Extruder\WObj:=Workobject_1;
MoveL RelTool (p1,35.000000,3.000000,17.287563,\Rx:=0.000000,\Ry:=-2.131683),vel1,zoneval,Extruder\WObj:=Workobject_1;
MoveL RelTool (p1,37.500000,3.000000,17.664646,\Rx:=0.000000,\Ry:=-1.262088),vel1,zoneval,Extruder\WObj:=Workobject_1;
MoveL RelTool (p1,40.000000,3.000000,17.903753,\Rx:=0.000000,\Ry:=-0.420073),vel1,zoneval,Extruder\WObj:=Workobject_1;
MoveL RelTool (p1,42.500000,3.000000,17.986264,\Rx:=0.000000,\Ry:=-0.285634),vel1,zoneval,Extruder\WObj:=Workobject_1;
MoveL RelTool (p1,45.000000,3.000000,17.937412,\Rx:=0.000000,\Ry:=0.382304),vel1,zoneval,Extruder\WObj:=Workobject_1;
MoveL RelTool (p1,47.500000,3.000000,17.749144,\Rx:=0.000000,\Ry:=1.180016),vel1,zoneval,Extruder\WObj:=Workobject_1;
MoveL RelTool (p1,50.000000,3.000000,17.427595,\Rx:=0.000000,\Ry:=2.025279),vel1,zoneval,Extruder\WObj:=Workobject_1;
MoveL RelTool (p1,52.500000,3.000000,16.955240,\Rx:=0.000000,\Ry:=2.916112),vel1,zoneval,Extruder\WObj:=Workobject_1;
MoveL RelTool (p1,55.000000,3.000000,16.310614,\Rx:=0.000000,\Ry:=3.853351),vel1,zoneval,Extruder\WObj:=Workobject_1;
MoveL RelTool (p1,57.500000,3.000000,15.462037,\Rx:=0.000000,\Ry:=4.827931),vel1,zoneval,Extruder\WObj:=Workobject_1;
MoveL RelTool (p1,60.000000,3.000000,14.358434,\Rx:=0.000000,\Ry:=5.885785),vel1,zoneval,Extruder\WObj:=Workobject_1;
MoveL RelTool (p1,62.500000,3.000000,12.916116,\Rx:=0.000000,\Ry:=8.188425),vel1,zoneval,Extruder\WObj:=Workobject_1;
MoveL RelTool (p1,65.000000,3.000000,10.800529,\Rx:=0.000000,\Ry:=10.986339),vel1,zoneval,Extruder\WObj:=Workobject_1;
MoveL RelTool (p1,67.500000,3.000000,8.322622,\Rx:=0.000000,\Ry:=4.473458),vel1,zoneval,Extruder\WObj:=Workobject_1;
MoveL RelTool (p1,70.000000,3.000000,8.000000,\Rx:=0.000000,\Ry:=-0.000000),vel1,zoneval,Extruder\WObj:=Workobject_1;
MoveL RelTool (p1,72.500000,3.000000,8.000000,\Rx:=0.000000,\Ry:=-0.000000),vel1,zoneval,Extruder\WObj:=Workobject_1;
MoveL RelTool (p1,75.000000,3.000000,8.000000,\Rx:=0.000000,\Ry:=-0.000000),vel1,zoneval,Extruder\WObj:=Workobject_1;
MoveL RelTool (p1,77.500000,3.000000,8.000000,\Rx:=0.000000,\Ry:=-0.000000),vel1,zoneval,Extruder\WObj:=Workobject_1;
MoveL RelTool (p1,80.000000,3.000000,8.000000,\Rx:=0.000000,\Ry:=-0.000000),vel1,zoneval,Extruder\WObj:=Workobject_1;
MoveL RelTool (p1,82.500000,3.000000,8.000000,\Rx:=0.000000,\Ry:=-0.000000),vel1,zoneval,Extruder\WObj:=Workobject_1;
MoveL RelTool (p1,80.500000,3.500000,8.000000,\Rx:=0.000000,\Ry:=0.000000),vel1,zoneval,Extruder\WObj:=Workobject_1;
MoveL RelTool (p1,78.000000,3.500000,8.000000,\Rx:=0.000000,\Ry:=0.000000),vel1,zoneval,Extruder\WObj:=Workobject_1;
MoveL RelTool (p1,75.500000,3.500000,8.000000,\Rx:=0.000000,\Ry:=0.000000),vel1,zoneval,Extruder\WObj:=Workobject_1;
MoveL RelTool (p1,73.000000,3.500000,8.000000,\Rx:=0.000000,\Ry:=0.000000),vel1,zoneval,Extruder\WObj:=Workobject_1;
MoveL RelTool (p1,70.500000,3.500000,8.000000,\Rx:=0.000000,\Ry:=0.000000),vel1,zoneval,Extruder\WObj:=Workobject_1;
MoveL RelTool (p1,68.000000,3.500000,8.139346,\Rx:=0.000000,\Ry:=4.473458),vel1,zoneval,Extruder\WObj:=Workobject_1;
MoveL RelTool (p1,65.500000,3.500000,10.217883,\Rx:=0.000000,\Ry:=10.977053),vel1,zoneval,Extruder\WObj:=Workobject_1;
MoveL RelTool (p1,63.000000,3.500000,12.542449,\Rx:=0.000000,\Ry:=8.189406),vel1,zoneval,Extruder\WObj:=Workobject_1;
MoveL RelTool (p1,60.500000,3.500000,14.109595,\Rx:=0.000000,\Ry:=5.885785),vel1,zoneval,Extruder\WObj:=Workobject_1;
MoveL RelTool (p1,58.000000,3.500000,15.263516,\Rx:=0.000000,\Ry:=4.827931),vel1,zoneval,Extruder\WObj:=Workobject_1;
MoveL RelTool (p1,55.500000,3.500000,16.155479,\Rx:=0.000000,\Ry:=3.853351),vel1,zoneval,Extruder\WObj:=Workobject_1;
MoveL RelTool (p1,53.000000,3.500000,16.838712,\Rx:=0.000000,\Ry:=2.916112),vel1,zoneval,Extruder\WObj:=Workobject_1;
MoveL RelTool (p1,50.500000,3.500000,17.347875,\Rx:=0.000000,\Ry:=2.025279),vel1,zoneval,Extruder\WObj:=Workobject_1;
MoveL RelTool (p1,48.000000,3.500000,17.703498,\Rx:=0.000000,\Ry:=1.180016),vel1,zoneval,Extruder\WObj:=Workobject_1;
MoveL RelTool (p1,45.500000,3.500000,17.923198,\Rx:=0.000000,\Ry:=0.382304),vel1,zoneval,Extruder\WObj:=Workobject_1;
MoveL RelTool (p1,43.000000,3.500000,17.998286,\Rx:=0.000000,\Ry:=-0.286534),vel1,zoneval,Extruder\WObj:=Workobject_1;
MoveL RelTool (p1,40.500000,3.500000,17.921023,\Rx:=0.000000,\Ry:=-0.420073),vel1,zoneval,Extruder\WObj:=Workobject_1;
MoveL RelTool (p1,38.000000,3.500000,17.715205,\Rx:=0.000000,\Ry:=-1.262088),vel1,zoneval,Extruder\WObj:=Workobject_1;
MoveL RelTool (p1,35.500000,3.500000,17.373079,\Rx:=0.000000,\Ry:=-2.131683),vel1,zoneval,Extruder\WObj:=Workobject_1;
MoveL RelTool (p1,33.000000,3.500000,16.879628,\Rx:=0.000000,\Ry:=-3.054804),vel1,zoneval,Extruder\WObj:=Workobject_1;
MoveL RelTool (p1,30.500000,3.500000,16.211616,\Rx:=0.000000,\Ry:=-4.018116),vel1,zoneval,Extruder\WObj:=Workobject_1;
MoveL RelTool (p1,28.000000,3.500000,15.331555,\Rx:=0.000000,\Ry:=-5.044928),vel1,zoneval,Extruder\WObj:=Workobject_1;
MoveL RelTool (p1,25.500000,3.500000,14.185704,\Rx:=0.000000,\Ry:=-6.198553),vel1,zoneval,Extruder\WObj:=Workobject_1;
MoveL RelTool (p1,23.000000,3.500000,12.670095,\Rx:=0.000000,\Ry:=-8.132708),vel1,zoneval,Extruder\WObj:=Workobject_1;
MoveL RelTool (p1,20.500000,3.500000,10.421902,\Rx:=0.000000,\Ry:=-11.182689),vel1,zoneval,Extruder\WObj:=Workobject_1;
MoveL RelTool (p1,18.000000,3.500000,8.180767,\Rx:=0.000000,\Ry:=-3.082616),vel1,zoneval,Extruder\WObj:=Workobject_1;
MoveL RelTool (p1,15.500000,3.500000,8.000000,\Rx:=0.000000,\Ry:=0.000000),vel1,zoneval,Extruder\WObj:=Workobject_1;
MoveL RelTool (p1,13.000000,3.500000,8.000000,\Rx:=0.000000,\Ry:=0.000000),vel1,zoneval,Extruder\WObj:=Workobject_1;
MoveL RelTool (p1,10.500000,3.500000,8.000000,\Rx:=0.000000,\Ry:=0.000000),vel1,zoneval,Extruder\WObj:=Workobject_1;
MoveL RelTool (p1,8.000000,3.500000,8.000000,\Rx:=0.000000,\Ry:=0.000000),vel1,zoneval,Extruder\WObj:=Workobject_1;
MoveL RelTool (p1,5.500000,3.500000,8.000000,\Rx:=0.000000,\Ry:=0.000000),vel1,zoneval,Extruder\WObj:=Workobject_1;
MoveL RelTool (p1,3.000000,3.500000,8.000000,\Rx:=0.000000,\Ry:=0.000000),vel1,zoneval,Extruder\WObj:=Workobject_1;
MoveL RelTool (p1,5.000000,4.000000,8.000000,\Rx:=0.000000,\Ry:=-0.000000),vel1,zoneval,Extruder\WObj:=Workobject_1;
MoveL RelTool (p1,7.500000,4.000000,8.000000,\Rx:=0.000000,\Ry:=-0.000000),vel1,zoneval,Extruder\WObj:=Workobject_1;
MoveL RelTool (p1,10.000000,4.000000,8.000000,\Rx:=0.000000,\Ry:=-0.000000),vel1,zoneval,Extruder\WObj:=Workobject_1;
MoveL RelTool (p1,12.500000,4.000000,8.000000,\Rx:=0.000000,\Ry:=-0.000000),vel1,zoneval,Extruder\WObj:=Workobject_1;
MoveL RelTool (p1,15.000000,4.000000,8.000000,\Rx:=0.000000,\Ry:=-0.000000),vel1,zoneval,Extruder\WObj:=Workobject_1;
MoveL RelTool (p1,17.500000,4.000000,8.057291,\Rx:=0.000000,\Ry:=-3.082616),vel1,zoneval,Extruder\WObj:=Workobject_1;
MoveL RelTool (p1,20.000000,4.000000,9.819463,\Rx:=0.000000,\Ry:=-11.184496),vel1,zoneval,Extruder\WObj:=Workobject_1;
MoveL RelTool (p1,22.500000,4.000000,12.299639,\Rx:=0.000000,\Ry:=-8.122785),vel1,zoneval,Extruder\WObj:=Workobject_1;
MoveL RelTool (p1,25.000000,4.000000,13.922240,\Rx:=0.000000,\Ry:=-6.198553),vel1,zoneval,Extruder\WObj:=Workobject_1;
MoveL RelTool (p1,27.500000,4.000000,15.122734,\Rx:=0.000000,\Ry:=-5.044928),vel1,zoneval,Extruder\WObj:=Workobject_1;
MoveL RelTool (p1,30.000000,4.000000,16.049016,\Rx:=0.000000,\Ry:=-4.018116),vel1,zoneval,Extruder\WObj:=Workobject_1;
MoveL RelTool (p1,32.500000,4.000000,16.757466,\Rx:=0.000000,\Ry:=-3.054804),vel1,zoneval,Extruder\WObj:=Workobject_1;
MoveL RelTool (p1,35.000000,4.000000,17.289591,\Rx:=0.000000,\Ry:=-2.131683),vel1,zoneval,Extruder\WObj:=Workobject_1;
MoveL RelTool (p1,37.500000,4.000000,17.666314,\Rx:=0.000000,\Ry:=-1.262088),vel1,zoneval,Extruder\WObj:=Workobject_1;
MoveL RelTool (p1,40.000000,4.000000,17.905288,\Rx:=0.000000,\Ry:=-0.420073),vel1,zoneval,Extruder\WObj:=Workobject_1;
MoveL RelTool (p1,42.500000,4.000000,17.987799,\Rx:=0.000000,\Ry:=-0.278595),vel1,zoneval,Extruder\WObj:=Workobject_1;
MoveL RelTool (p1,45.000000,4.000000,17.939018,\Rx:=0.000000,\Ry:=0.382304),vel1,zoneval,Extruder\WObj:=Workobject_1;
MoveL RelTool (p1,47.500000,4.000000,17.750796,\Rx:=0.000000,\Ry:=1.180016),vel1,zoneval,Extruder\WObj:=Workobject_1;
MoveL RelTool (p1,50.000000,4.000000,17.428576,\Rx:=0.000000,\Ry:=2.025279),vel1,zoneval,Extruder\WObj:=Workobject_1;
MoveL RelTool (p1,52.500000,4.000000,16.955306,\Rx:=0.000000,\Ry:=2.916112),vel1,zoneval,Extruder\WObj:=Workobject_1;
MoveL RelTool (p1,55.000000,4.000000,16.312577,\Rx:=0.000000,\Ry:=3.853351),vel1,zoneval,Extruder\WObj:=Workobject_1;
MoveL RelTool (p1,57.500000,4.000000,15.463463,\Rx:=0.000000,\Ry:=4.827931),vel1,zoneval,Extruder\WObj:=Workobject_1;
MoveL RelTool (p1,60.000000,4.000000,14.359033,\Rx:=0.000000,\Ry:=5.885785),vel1,zoneval,Extruder\WObj:=Workobject_1;
MoveL RelTool (p1,62.500000,4.000000,12.918302,\Rx:=0.000000,\Ry:=8.190386),vel1,zoneval,Extruder\WObj:=Workobject_1;
MoveL RelTool (p1,65.000000,4.000000,10.801823,\Rx:=0.000000,\Ry:=10.967752),vel1,zoneval,Extruder\WObj:=Workobject_1;
MoveL RelTool (p1,67.500000,4.000000,8.322622,\Rx:=0.000000,\Ry:=4.473458),vel1,zoneval,Extruder\WObj:=Workobject_1;
MoveL RelTool (p1,70.000000,4.000000,8.000000,\Rx:=0.000000,\Ry:=-0.000000),vel1,zoneval,Extruder\WObj:=Workobject_1;
MoveL RelTool (p1,72.500000,4.000000,8.000000,\Rx:=0.000000,\Ry:=-0.000000),vel1,zoneval,Extruder\WObj:=Workobject_1;
MoveL RelTool (p1,75.000000,4.000000,8.000000,\Rx:=0.000000,\Ry:=-0.000000),vel1,zoneval,Extruder\WObj:=Workobject_1;
MoveL RelTool (p1,77.500000,4.000000,8.000000,\Rx:=0.000000,\Ry:=-0.000000),vel1,zoneval,Extruder\WObj:=Workobject_1;
MoveL RelTool (p1,80.000000,4.000000,8.000000,\Rx:=0.000000,\Ry:=-0.000000),vel1,zoneval,Extruder\WObj:=Workobject_1;
MoveL RelTool (p1,82.500000,4.000000,8.000000,\Rx:=0.000000,\Ry:=-0.000000),vel1,zoneval,Extruder\WObj:=Workobject_1;
MoveL RelTool (p1,80.500000,4.500000,8.000000,\Rx:=0.000000,\Ry:=0.000000),vel1,zoneval,Extruder\WObj:=Workobject_1;
MoveL RelTool (p1,78.000000,4.500000,8.000000,\Rx:=0.000000,\Ry:=0.000000),vel1,zoneval,Extruder\WObj:=Workobject_1;
MoveL RelTool (p1,75.500000,4.500000,8.000000,\Rx:=0.000000,\Ry:=0.000000),vel1,zoneval,Extruder\WObj:=Workobject_1;
MoveL RelTool (p1,73.000000,4.500000,8.000000,\Rx:=0.000000,\Ry:=0.000000),vel1,zoneval,Extruder\WObj:=Workobject_1;
MoveL RelTool (p1,70.500000,4.500000,8.000000,\Rx:=0.000000,\Ry:=0.000000),vel1,zoneval,Extruder\WObj:=Workobject_1;
MoveL RelTool (p1,68.000000,4.500000,8.139346,\Rx:=0.000000,\Ry:=4.473458),vel1,zoneval,Extruder\WObj:=Workobject_1;
MoveL RelTool (p1,65.500000,4.500000,10.220900,\Rx:=0.000000,\Ry:=10.958434),vel1,zoneval,Extruder\WObj:=Workobject_1;
MoveL RelTool (p1,63.000000,4.500000,12.544514,\Rx:=0.000000,\Ry:=8.176295),vel1,zoneval,Extruder\WObj:=Workobject_1;
MoveL RelTool (p1,60.500000,4.500000,14.110193,\Rx:=0.000000,\Ry:=5.885785),vel1,zoneval,Extruder\WObj:=Workobject_1;
MoveL RelTool (p1,58.000000,4.500000,15.264942,\Rx:=0.000000,\Ry:=4.827931),vel1,zoneval,Extruder\WObj:=Workobject_1;
MoveL RelTool (p1,55.500000,4.500000,16.157442,\Rx:=0.000000,\Ry:=3.853351),vel1,zoneval,Extruder\WObj:=Workobject_1;
MoveL RelTool (p1,53.000000,4.500000,16.838778,\Rx:=0.000000,\Ry:=2.916112),vel1,zoneval,Extruder\WObj:=Workobject_1;
MoveL RelTool (p1,50.500000,4.500000,17.348856,\Rx:=0.000000,\Ry:=2.025279),vel1,zoneval,Extruder\WObj:=Workobject_1;
MoveL RelTool (p1,48.000000,4.500000,17.705149,\Rx:=0.000000,\Ry:=1.180016),vel1,zoneval,Extruder\WObj:=Workobject_1;
MoveL RelTool (p1,45.500000,4.500000,17.924804,\Rx:=0.000000,\Ry:=0.382304),vel1,zoneval,Extruder\WObj:=Workobject_1;
MoveL RelTool (p1,43.000000,4.500000,17.998490,\Rx:=0.000000,\Ry:=-0.252662),vel1,zoneval,Extruder\WObj:=Workobject_1;
MoveL RelTool (p1,40.500000,4.500000,17.922558,\Rx:=0.000000,\Ry:=-0.420073),vel1,zoneval,Extruder\WObj:=Workobject_1;
MoveL RelTool (p1,38.000000,4.500000,17.716873,\Rx:=0.000000,\Ry:=-1.262088),vel1,zoneval,Extruder\WObj:=Workobject_1;
MoveL RelTool (p1,35.500000,4.500000,17.375106,\Rx:=0.000000,\Ry:=-2.131683),vel1,zoneval,Extruder\WObj:=Workobject_1;
MoveL RelTool (p1,33.000000,4.500000,16.879940,\Rx:=0.000000,\Ry:=-3.054804),vel1,zoneval,Extruder\WObj:=Workobject_1;
MoveL RelTool (p1,30.500000,4.500000,16.212910,\Rx:=0.000000,\Ry:=-4.018116),vel1,zoneval,Extruder\WObj:=Workobject_1;
MoveL RelTool (p1,28.000000,4.500000,15.332266,\Rx:=0.000000,\Ry:=-5.044928),vel1,zoneval,Extruder\WObj:=Workobject_1;
MoveL RelTool (p1,25.500000,4.500000,14.188104,\Rx:=0.000000,\Ry:=-6.198553),vel1,zoneval,Extruder\WObj:=Workobject_1;
MoveL RelTool (p1,23.000000,4.500000,12.670563,\Rx:=0.000000,\Ry:=-8.112850),vel1,zoneval,Extruder\WObj:=Workobject_1;
MoveL RelTool (p1,20.500000,4.500000,10.422825,\Rx:=0.000000,\Ry:=-11.186304),vel1,zoneval,Extruder\WObj:=Workobject_1;
MoveL RelTool (p1,18.000000,4.500000,8.180767,\Rx:=0.000000,\Ry:=-3.082616),vel1,zoneval,Extruder\WObj:=Workobject_1;
MoveL RelTool (p1,15.500000,4.500000,8.000000,\Rx:=0.000000,\Ry:=0.000000),vel1,zoneval,Extruder\WObj:=Workobject_1;
MoveL RelTool (p1,13.000000,4.500000,8.000000,\Rx:=0.000000,\Ry:=0.000000),vel1,zoneval,Extruder\WObj:=Workobject_1;
MoveL RelTool (p1,10.500000,4.500000,8.000000,\Rx:=0.000000,\Ry:=0.000000),vel1,zoneval,Extruder\WObj:=Workobject_1;
MoveL RelTool (p1,8.000000,4.500000,8.000000,\Rx:=0.000000,\Ry:=0.000000),vel1,zoneval,Extruder\WObj:=Workobject_1;
MoveL RelTool (p1,5.500000,4.500000,8.000000,\Rx:=0.000000,\Ry:=0.000000),vel1,zoneval,Extruder\WObj:=Workobject_1;
MoveL RelTool (p1,3.000000,4.500000,8.000000,\Rx:=0.000000,\Ry:=0.000000),vel1,zoneval,Extruder\WObj:=Workobject_1;
MoveL RelTool (p1,5.000000,5.000000,8.000000,\Rx:=0.000000,\Ry:=-0.000000),vel1,zoneval,Extruder\WObj:=Workobject_1;
MoveL RelTool (p1,7.500000,5.000000,8.000000,\Rx:=0.000000,\Ry:=-0.000000),vel1,zoneval,Extruder\WObj:=Workobject_1;
MoveL RelTool (p1,10.000000,5.000000,8.000000,\Rx:=0.000000,\Ry:=-0.000000),vel1,zoneval,Extruder\WObj:=Workobject_1;
MoveL RelTool (p1,12.500000,5.000000,8.000000,\Rx:=0.000000,\Ry:=-0.000000),vel1,zoneval,Extruder\WObj:=Workobject_1;
MoveL RelTool (p1,15.000000,5.000000,8.000000,\Rx:=0.000000,\Ry:=-0.000000),vel1,zoneval,Extruder\WObj:=Workobject_1;
MoveL RelTool (p1,17.500000,5.000000,8.057291,\Rx:=0.000000,\Ry:=-3.082616),vel1,zoneval,Extruder\WObj:=Workobject_1;
MoveL RelTool (p1,20.000000,5.000000,9.820038,\Rx:=0.000000,\Ry:=-11.188110),vel1,zoneval,Extruder\WObj:=Workobject_1;
MoveL RelTool (p1,22.500000,5.000000,12.301315,\Rx:=0.000000,\Ry:=-8.102905),vel1,zoneval,Extruder\WObj:=Workobject_1;
MoveL RelTool (p1,25.000000,5.000000,13.924640,\Rx:=0.000000,\Ry:=-6.198553),vel1,zoneval,Extruder\WObj:=Workobject_1;
MoveL RelTool (p1,27.500000,5.000000,15.123444,\Rx:=0.000000,\Ry:=-5.044928),vel1,zoneval,Extruder\WObj:=Workobject_1;
MoveL RelTool (p1,30.000000,5.000000,16.050310,\Rx:=0.000000,\Ry:=-4.018116),vel1,zoneval,Extruder\WObj:=Workobject_1;
MoveL RelTool (p1,32.500000,5.000000,16.757778,\Rx:=0.000000,\Ry:=-3.054804),vel1,zoneval,Extruder\WObj:=Workobject_1;
MoveL RelTool (p1,35.000000,5.000000,17.291618,\Rx:=0.000000,\Ry:=-2.131683),vel1,zoneval,Extruder\WObj:=Workobject_1;
MoveL RelTool (p1,37.500000,5.000000,17.667982,\Rx:=0.000000,\Ry:=-1.262088),vel1,zoneval,Extruder\WObj:=Workobject_1;
MoveL RelTool (p1,40.000000,5.000000,17.906823,\Rx:=0.000000,\Ry:=-0.420073),vel1,zoneval,Extruder\WObj:=Workobject_1;
MoveL RelTool (p1,42.500000,5.000000,17.989334,\Rx:=0.000000,\Ry:=-0.226726),vel1,zoneval,Extruder\WObj:=Workobject_1;
MoveL RelTool (p1,45.000000,5.000000,17.940624,\Rx:=0.000000,\Ry:=0.394040),vel1,zoneval,Extruder\WObj:=Workobject_1;
MoveL RelTool (p1,47.500000,5.000000,17.752447,\Rx:=0.000000,\Ry:=1.180016),vel1,zoneval,Extruder\WObj:=Workobject_1;
MoveL RelTool (p1,50.000000,5.000000,17.429557,\Rx:=0.000000,\Ry:=2.025279),vel1,zoneval,Extruder\WObj:=Workobject_1;
MoveL RelTool (p1,52.500000,5.000000,16.955372,\Rx:=0.000000,\Ry:=2.916112),vel1,zoneval,Extruder\WObj:=Workobject_1;
MoveL RelTool (p1,55.000000,5.000000,16.314540,\Rx:=0.000000,\Ry:=3.853351),vel1,zoneval,Extruder\WObj:=Workobject_1;
MoveL RelTool (p1,57.500000,5.000000,15.464889,\Rx:=0.000000,\Ry:=4.827931),vel1,zoneval,Extruder\WObj:=Workobject_1;
MoveL RelTool (p1,60.000000,5.000000,14.359631,\Rx:=0.000000,\Ry:=5.885785),vel1,zoneval,Extruder\WObj:=Workobject_1;
MoveL RelTool (p1,62.500000,5.000000,12.918262,\Rx:=0.000000,\Ry:=8.156002),vel1,zoneval,Extruder\WObj:=Workobject_1;
MoveL RelTool (p1,65.000000,5.000000,10.803116,\Rx:=0.000000,\Ry:=10.949101),vel1,zoneval,Extruder\WObj:=Workobject_1;
MoveL RelTool (p1,67.500000,5.000000,8.322622,\Rx:=0.000000,\Ry:=4.473458),vel1,zoneval,Extruder\WObj:=Workobject_1;
MoveL RelTool (p1,70.000000,5.000000,8.000000,\Rx:=0.000000,\Ry:=-0.000000),vel1,zoneval,Extruder\WObj:=Workobject_1;
MoveL RelTool (p1,72.500000,5.000000,8.000000,\Rx:=0.000000,\Ry:=-0.000000),vel1,zoneval,Extruder\WObj:=Workobject_1;
MoveL RelTool (p1,75.000000,5.000000,8.000000,\Rx:=0.000000,\Ry:=-0.000000),vel1,zoneval,Extruder\WObj:=Workobject_1;
MoveL RelTool (p1,77.500000,5.000000,8.000000,\Rx:=0.000000,\Ry:=-0.000000),vel1,zoneval,Extruder\WObj:=Workobject_1;
MoveL RelTool (p1,80.000000,5.000000,8.000000,\Rx:=0.000000,\Ry:=-0.000000),vel1,zoneval,Extruder\WObj:=Workobject_1;
MoveL RelTool (p1,82.500000,5.000000,8.000000,\Rx:=0.000000,\Ry:=-0.000000),vel1,zoneval,Extruder\WObj:=Workobject_1;
MoveL RelTool (p1,80.500000,5.500000,8.000000,\Rx:=0.000000,\Ry:=0.000000),vel1,zoneval,Extruder\WObj:=Workobject_1;
MoveL RelTool (p1,78.000000,5.500000,8.000000,\Rx:=0.000000,\Ry:=0.000000),vel1,zoneval,Extruder\WObj:=Workobject_1;
MoveL RelTool (p1,75.500000,5.500000,8.000000,\Rx:=0.000000,\Ry:=0.000000),vel1,zoneval,Extruder\WObj:=Workobject_1;
MoveL RelTool (p1,73.000000,5.500000,8.000000,\Rx:=0.000000,\Ry:=0.000000),vel1,zoneval,Extruder\WObj:=Workobject_1;
MoveL RelTool (p1,70.500000,5.500000,8.000000,\Rx:=0.000000,\Ry:=0.000000),vel1,zoneval,Extruder\WObj:=Workobject_1;
MoveL RelTool (p1,68.000000,5.500000,8.139346,\Rx:=0.000000,\Ry:=4.473458),vel1,zoneval,Extruder\WObj:=Workobject_1;
MoveL RelTool (p1,65.500000,5.500000,10.223917,\Rx:=0.000000,\Ry:=10.939752),vel1,zoneval,Extruder\WObj:=Workobject_1;
MoveL RelTool (p1,63.000000,5.500000,12.546579,\Rx:=0.000000,\Ry:=8.135661),vel1,zoneval,Extruder\WObj:=Workobject_1;
MoveL RelTool (p1,60.500000,5.500000,14.110792,\Rx:=0.000000,\Ry:=5.885785),vel1,zoneval,Extruder\WObj:=Workobject_1;
MoveL RelTool (p1,58.000000,5.500000,15.266367,\Rx:=0.000000,\Ry:=4.827931),vel1,zoneval,Extruder\WObj:=Workobject_1;
MoveL RelTool (p1,55.500000,5.500000,16.159405,\Rx:=0.000000,\Ry:=3.853351),vel1,zoneval,Extruder\WObj:=Workobject_1;
MoveL RelTool (p1,53.000000,5.500000,16.838844,\Rx:=0.000000,\Ry:=2.916112),vel1,zoneval,Extruder\WObj:=Workobject_1;
MoveL RelTool (p1,50.500000,5.500000,17.349838,\Rx:=0.000000,\Ry:=2.025279),vel1,zoneval,Extruder\WObj:=Workobject_1;
MoveL RelTool (p1,48.000000,5.500000,17.706801,\Rx:=0.000000,\Ry:=1.180016),vel1,zoneval,Extruder\WObj:=Workobject_1;
MoveL RelTool (p1,45.500000,5.500000,17.924970,\Rx:=0.000000,\Ry:=0.418928),vel1,zoneval,Extruder\WObj:=Workobject_1;
MoveL RelTool (p1,43.000000,5.500000,17.997987,\Rx:=0.000000,\Ry:=-0.202149),vel1,zoneval,Extruder\WObj:=Workobject_1;
MoveL RelTool (p1,40.500000,5.500000,17.924093,\Rx:=0.000000,\Ry:=-0.433388),vel1,zoneval,Extruder\WObj:=Workobject_1;
MoveL RelTool (p1,38.000000,5.500000,17.718541,\Rx:=0.000000,\Ry:=-1.262088),vel1,zoneval,Extruder\WObj:=Workobject_1;
MoveL RelTool (p1,35.500000,5.500000,17.377134,\Rx:=0.000000,\Ry:=-2.131683),vel1,zoneval,Extruder\WObj:=Workobject_1;
MoveL RelTool (p1,33.000000,5.500000,16.880251,\Rx:=0.000000,\Ry:=-3.054804),vel1,zoneval,Extruder\WObj:=Workobject_1;
MoveL RelTool (p1,30.500000,5.500000,16.214204,\Rx:=0.000000,\Ry:=-4.018116),vel1,zoneval,Extruder\WObj:=Workobject_1;
MoveL RelTool (p1,28.000000,5.500000,15.332976,\Rx:=0.000000,\Ry:=-5.044928),vel1,zoneval,Extruder\WObj:=Workobject_1;
MoveL RelTool (p1,25.500000,5.500000,14.190503,\Rx:=0.000000,\Ry:=-6.198553),vel1,zoneval,Extruder\WObj:=Workobject_1;
MoveL RelTool (p1,23.000000,5.500000,12.671773,\Rx:=0.000000,\Ry:=-8.105191),vel1,zoneval,Extruder\WObj:=Workobject_1;
MoveL RelTool (p1,20.500000,5.500000,10.423747,\Rx:=0.000000,\Ry:=-11.189916),vel1,zoneval,Extruder\WObj:=Workobject_1;
MoveL RelTool (p1,18.000000,5.500000,8.180767,\Rx:=0.000000,\Ry:=-3.082616),vel1,zoneval,Extruder\WObj:=Workobject_1;
MoveL RelTool (p1,15.500000,5.500000,8.000000,\Rx:=0.000000,\Ry:=0.000000),vel1,zoneval,Extruder\WObj:=Workobject_1;
MoveL RelTool (p1,13.000000,5.500000,8.000000,\Rx:=0.000000,\Ry:=0.000000),vel1,zoneval,Extruder\WObj:=Workobject_1;
MoveL RelTool (p1,10.500000,5.500000,8.000000,\Rx:=0.000000,\Ry:=0.000000),vel1,zoneval,Extruder\WObj:=Workobject_1;
MoveL RelTool (p1,8.000000,5.500000,8.000000,\Rx:=0.000000,\Ry:=0.000000),vel1,zoneval,Extruder\WObj:=Workobject_1;
MoveL RelTool (p1,5.500000,5.500000,8.000000,\Rx:=0.000000,\Ry:=0.000000),vel1,zoneval,Extruder\WObj:=Workobject_1;
MoveL RelTool (p1,3.000000,5.500000,8.000000,\Rx:=0.000000,\Ry:=0.000000),vel1,zoneval,Extruder\WObj:=Workobject_1;
MoveL RelTool (p1,5.000000,6.000000,8.000000,\Rx:=0.000000,\Ry:=-0.000000),vel1,zoneval,Extruder\WObj:=Workobject_1;
MoveL RelTool (p1,7.500000,6.000000,8.000000,\Rx:=0.000000,\Ry:=-0.000000),vel1,zoneval,Extruder\WObj:=Workobject_1;
MoveL RelTool (p1,10.000000,6.000000,8.000000,\Rx:=0.000000,\Ry:=-0.000000),vel1,zoneval,Extruder\WObj:=Workobject_1;
MoveL RelTool (p1,12.500000,6.000000,8.000000,\Rx:=0.000000,\Ry:=-0.000000),vel1,zoneval,Extruder\WObj:=Workobject_1;
MoveL RelTool (p1,15.000000,6.000000,8.000000,\Rx:=0.000000,\Ry:=-0.000000),vel1,zoneval,Extruder\WObj:=Workobject_1;
MoveL RelTool (p1,17.500000,6.000000,8.057291,\Rx:=0.000000,\Ry:=-3.082616),vel1,zoneval,Extruder\WObj:=Workobject_1;
MoveL RelTool (p1,20.000000,6.000000,9.820612,\Rx:=0.000000,\Ry:=-11.191722),vel1,zoneval,Extruder\WObj:=Workobject_1;
MoveL RelTool (p1,22.500000,6.000000,12.302990,\Rx:=0.000000,\Ry:=-8.119028),vel1,zoneval,Extruder\WObj:=Workobject_1;
MoveL RelTool (p1,25.000000,6.000000,13.927039,\Rx:=0.000000,\Ry:=-6.198553),vel1,zoneval,Extruder\WObj:=Workobject_1;
MoveL RelTool (p1,27.500000,6.000000,15.124154,\Rx:=0.000000,\Ry:=-5.044928),vel1,zoneval,Extruder\WObj:=Workobject_1;
MoveL RelTool (p1,30.000000,6.000000,16.051604,\Rx:=0.000000,\Ry:=-4.018116),vel1,zoneval,Extruder\WObj:=Workobject_1;
MoveL RelTool (p1,32.500000,6.000000,16.758089,\Rx:=0.000000,\Ry:=-3.054804),vel1,zoneval,Extruder\WObj:=Workobject_1;
MoveL RelTool (p1,35.000000,6.000000,17.293645,\Rx:=0.000000,\Ry:=-2.131683),vel1,zoneval,Extruder\WObj:=Workobject_1;
MoveL RelTool (p1,37.500000,6.000000,17.669649,\Rx:=0.000000,\Ry:=-1.262088),vel1,zoneval,Extruder\WObj:=Workobject_1;
MoveL RelTool (p1,40.000000,6.000000,17.906744,\Rx:=0.000000,\Ry:=-0.461125),vel1,zoneval,Extruder\WObj:=Workobject_1;
MoveL RelTool (p1,42.500000,6.000000,17.990481,\Rx:=0.000000,\Ry:=-0.184751),vel1,zoneval,Extruder\WObj:=Workobject_1;
MoveL RelTool (p1,45.000000,6.000000,17.942230,\Rx:=0.000000,\Ry:=0.443814),vel1,zoneval,Extruder\WObj:=Workobject_1;
MoveL RelTool (p1,47.500000,6.000000,17.754099,\Rx:=0.000000,\Ry:=1.180016),vel1,zoneval,Extruder\WObj:=Workobject_1;
MoveL RelTool (p1,50.000000,6.000000,17.430539,\Rx:=0.000000,\Ry:=2.025279),vel1,zoneval,Extruder\WObj:=Workobject_1;
MoveL RelTool (p1,52.500000,6.000000,16.955437,\Rx:=0.000000,\Ry:=2.916112),vel1,zoneval,Extruder\WObj:=Workobject_1;
MoveL RelTool (p1,55.000000,6.000000,16.316503,\Rx:=0.000000,\Ry:=3.853351),vel1,zoneval,Extruder\WObj:=Workobject_1;
MoveL RelTool (p1,57.500000,6.000000,15.466314,\Rx:=0.000000,\Ry:=4.827931),vel1,zoneval,Extruder\WObj:=Workobject_1;
MoveL RelTool (p1,60.000000,6.000000,14.360230,\Rx:=0.000000,\Ry:=5.885785),vel1,zoneval,Extruder\WObj:=Workobject_1;
MoveL RelTool (p1,62.500000,6.000000,12.917845,\Rx:=0.000000,\Ry:=8.115271),vel1,zoneval,Extruder\WObj:=Workobject_1;
MoveL RelTool (p1,65.000000,6.000000,10.804410,\Rx:=0.000000,\Ry:=10.930386),vel1,zoneval,Extruder\WObj:=Workobject_1;
MoveL RelTool (p1,67.500000,6.000000,8.322622,\Rx:=0.000000,\Ry:=4.473458),vel1,zoneval,Extruder\WObj:=Workobject_1;
MoveL RelTool (p1,70.000000,6.000000,8.000000,\Rx:=0.000000,\Ry:=-0.000000),vel1,zoneval,Extruder\WObj:=Workobject_1;
MoveL RelTool (p1,72.500000,6.000000,8.000000,\Rx:=0.000000,\Ry:=-0.000000),vel1,zoneval,Extruder\WObj:=Workobject_1;
MoveL RelTool (p1,75.000000,6.000000,8.000000,\Rx:=0.000000,\Ry:=-0.000000),vel1,zoneval,Extruder\WObj:=Workobject_1;
MoveL RelTool (p1,77.500000,6.000000,8.000000,\Rx:=0.000000,\Ry:=-0.000000),vel1,zoneval,Extruder\WObj:=Workobject_1;
MoveL RelTool (p1,80.000000,6.000000,8.000000,\Rx:=0.000000,\Ry:=-0.000000),vel1,zoneval,Extruder\WObj:=Workobject_1;
MoveL RelTool (p1,82.500000,6.000000,8.000000,\Rx:=0.000000,\Ry:=-0.000000),vel1,zoneval,Extruder\WObj:=Workobject_1;
MoveL RelTool (p1,80.500000,6.500000,8.000000,\Rx:=0.000000,\Ry:=0.000000),vel1,zoneval,Extruder\WObj:=Workobject_1;
MoveL RelTool (p1,78.000000,6.500000,8.000000,\Rx:=0.000000,\Ry:=0.000000),vel1,zoneval,Extruder\WObj:=Workobject_1;
MoveL RelTool (p1,75.500000,6.500000,8.000000,\Rx:=0.000000,\Ry:=0.000000),vel1,zoneval,Extruder\WObj:=Workobject_1;
MoveL RelTool (p1,73.000000,6.500000,8.000000,\Rx:=0.000000,\Ry:=0.000000),vel1,zoneval,Extruder\WObj:=Workobject_1;
MoveL RelTool (p1,70.500000,6.500000,8.000000,\Rx:=0.000000,\Ry:=0.000000),vel1,zoneval,Extruder\WObj:=Workobject_1;
MoveL RelTool (p1,68.000000,6.500000,8.139346,\Rx:=0.000000,\Ry:=4.473458),vel1,zoneval,Extruder\WObj:=Workobject_1;
MoveL RelTool (p1,65.500000,6.500000,10.226934,\Rx:=0.000000,\Ry:=10.921005),vel1,zoneval,Extruder\WObj:=Workobject_1;
MoveL RelTool (p1,63.000000,6.500000,12.548644,\Rx:=0.000000,\Ry:=8.094833),vel1,zoneval,Extruder\WObj:=Workobject_1;
MoveL RelTool (p1,60.500000,6.500000,14.111391,\Rx:=0.000000,\Ry:=5.885785),vel1,zoneval,Extruder\WObj:=Workobject_1;
MoveL RelTool (p1,58.000000,6.500000,15.267793,\Rx:=0.000000,\Ry:=4.827931),vel1,zoneval,Extruder\WObj:=Workobject_1;
MoveL RelTool (p1,55.500000,6.500000,16.161368,\Rx:=0.000000,\Ry:=3.853351),vel1,zoneval,Extruder\WObj:=Workobject_1;
MoveL RelTool (p1,53.000000,6.500000,16.838910,\Rx:=0.000000,\Ry:=2.916112),vel1,zoneval,Extruder\WObj:=Workobject_1;
MoveL RelTool (p1,50.500000,6.500000,17.350819,\Rx:=0.000000,\Ry:=2.025279),vel1,zoneval,Extruder\WObj:=Workobject_1;
MoveL RelTool (p1,48.000000,6.500000,17.708452,\Rx:=0.000000,\Ry:=1.180016),vel1,zoneval,Extruder\WObj:=Workobject_1;
MoveL RelTool (p1,45.500000,6.500000,17.924619,\Rx:=0.000000,\Ry:=0.468696),vel1,zoneval,Extruder\WObj:=Workobject_1;
MoveL RelTool (p1,43.000000,6.500000,17.997485,\Rx:=0.000000,\Ry:=-0.167353),vel1,zoneval,Extruder\WObj:=Workobject_1;
MoveL RelTool (p1,40.500000,6.500000,17.925628,\Rx:=0.000000,\Ry:=-0.488858),vel1,zoneval,Extruder\WObj:=Workobject_1;
MoveL RelTool (p1,38.000000,6.500000,17.720208,\Rx:=0.000000,\Ry:=-1.262088),vel1,zoneval,Extruder\WObj:=Workobject_1;
MoveL RelTool (p1,35.500000,6.500000,17.379161,\Rx:=0.000000,\Ry:=-2.131683),vel1,zoneval,Extruder\WObj:=Workobject_1;
MoveL RelTool (p1,33.000000,6.500000,16.880563,\Rx:=0.000000,\Ry:=-3.054804),vel1,zoneval,Extruder\WObj:=Workobject_1;
MoveL RelTool (p1,30.500000,6.500000,16.215498,\Rx:=0.000000,\Ry:=-4.018116),vel1,zoneval,Extruder\WObj:=Workobject_1;
MoveL RelTool (p1,28.000000,6.500000,15.333686,\Rx:=0.000000,\Ry:=-5.044928),vel1,zoneval,Extruder\WObj:=Workobject_1;
MoveL RelTool (p1,25.500000,6.500000,14.192902,\Rx:=0.000000,\Ry:=-6.198553),vel1,zoneval,Extruder\WObj:=Workobject_1;
MoveL RelTool (p1,23.000000,6.500000,12.675131,\Rx:=0.000000,\Ry:=-8.132843),vel1,zoneval,Extruder\WObj:=Workobject_1;
MoveL RelTool (p1,20.500000,6.500000,10.424670,\Rx:=0.000000,\Ry:=-11.193527),vel1,zoneval,Extruder\WObj:=Workobject_1;
MoveL RelTool (p1,18.000000,6.500000,8.180767,\Rx:=0.000000,\Ry:=-3.082616),vel1,zoneval,Extruder\WObj:=Workobject_1;
MoveL RelTool (p1,15.500000,6.500000,8.000000,\Rx:=0.000000,\Ry:=0.000000),vel1,zoneval,Extruder\WObj:=Workobject_1;
MoveL RelTool (p1,13.000000,6.500000,8.000000,\Rx:=0.000000,\Ry:=0.000000),vel1,zoneval,Extruder\WObj:=Workobject_1;
MoveL RelTool (p1,10.500000,6.500000,8.000000,\Rx:=0.000000,\Ry:=0.000000),vel1,zoneval,Extruder\WObj:=Workobject_1;
MoveL RelTool (p1,8.000000,6.500000,8.000000,\Rx:=0.000000,\Ry:=0.000000),vel1,zoneval,Extruder\WObj:=Workobject_1;
MoveL RelTool (p1,5.500000,6.500000,8.000000,\Rx:=0.000000,\Ry:=0.000000),vel1,zoneval,Extruder\WObj:=Workobject_1;
MoveL RelTool (p1,3.000000,6.500000,8.000000,\Rx:=0.000000,\Ry:=0.000000),vel1,zoneval,Extruder\WObj:=Workobject_1;
MoveL RelTool (p1,5.000000,7.000000,8.000000,\Rx:=0.000000,\Ry:=-0.000000),vel1,zoneval,Extruder\WObj:=Workobject_1;
MoveL RelTool (p1,7.500000,7.000000,8.000000,\Rx:=0.000000,\Ry:=-0.000000),vel1,zoneval,Extruder\WObj:=Workobject_1;
MoveL RelTool (p1,10.000000,7.000000,8.000000,\Rx:=0.000000,\Ry:=-0.000000),vel1,zoneval,Extruder\WObj:=Workobject_1;
MoveL RelTool (p1,12.500000,7.000000,8.000000,\Rx:=0.000000,\Ry:=-0.000000),vel1,zoneval,Extruder\WObj:=Workobject_1;
MoveL RelTool (p1,15.000000,7.000000,8.000000,\Rx:=0.000000,\Ry:=-0.000000),vel1,zoneval,Extruder\WObj:=Workobject_1;
MoveL RelTool (p1,17.500000,7.000000,8.057291,\Rx:=0.000000,\Ry:=-3.082616),vel1,zoneval,Extruder\WObj:=Workobject_1;
MoveL RelTool (p1,20.000000,7.000000,9.821186,\Rx:=0.000000,\Ry:=-11.195331),vel1,zoneval,Extruder\WObj:=Workobject_1;
MoveL RelTool (p1,22.500000,7.000000,12.304666,\Rx:=0.000000,\Ry:=-8.146636),vel1,zoneval,Extruder\WObj:=Workobject_1;
MoveL RelTool (p1,25.000000,7.000000,13.929438,\Rx:=0.000000,\Ry:=-6.198553),vel1,zoneval,Extruder\WObj:=Workobject_1;
MoveL RelTool (p1,27.500000,7.000000,15.124865,\Rx:=0.000000,\Ry:=-5.044928),vel1,zoneval,Extruder\WObj:=Workobject_1;
MoveL RelTool (p1,30.000000,7.000000,16.052898,\Rx:=0.000000,\Ry:=-4.018116),vel1,zoneval,Extruder\WObj:=Workobject_1;
MoveL RelTool (p1,32.500000,7.000000,16.758401,\Rx:=0.000000,\Ry:=-3.054804),vel1,zoneval,Extruder\WObj:=Workobject_1;
MoveL RelTool (p1,35.000000,7.000000,17.295673,\Rx:=0.000000,\Ry:=-2.131683),vel1,zoneval,Extruder\WObj:=Workobject_1;
MoveL RelTool (p1,37.500000,7.000000,17.671317,\Rx:=0.000000,\Ry:=-1.262088),vel1,zoneval,Extruder\WObj:=Workobject_1;
MoveL RelTool (p1,40.000000,7.000000,17.906098,\Rx:=0.000000,\Ry:=-0.516586),vel1,zoneval,Extruder\WObj:=Workobject_1;
MoveL RelTool (p1,42.500000,7.000000,17.991345,\Rx:=0.000000,\Ry:=-0.149953),vel1,zoneval,Extruder\WObj:=Workobject_1;
MoveL RelTool (p1,45.000000,7.000000,17.943836,\Rx:=0.000000,\Ry:=0.493574),vel1,zoneval,Extruder\WObj:=Workobject_1;
MoveL RelTool (p1,47.500000,7.000000,17.755750,\Rx:=0.000000,\Ry:=1.180016),vel1,zoneval,Extruder\WObj:=Workobject_1;
MoveL RelTool (p1,50.000000,7.000000,17.431520,\Rx:=0.000000,\Ry:=2.025279),vel1,zoneval,Extruder\WObj:=Workobject_1;
MoveL RelTool (p1,52.500000,7.000000,16.955503,\Rx:=0.000000,\Ry:=2.916112),vel1,zoneval,Extruder\WObj:=Workobject_1;
MoveL RelTool (p1,55.000000,7.000000,16.318466,\Rx:=0.000000,\Ry:=3.853351),vel1,zoneval,Extruder\WObj:=Workobject_1;
MoveL RelTool (p1,57.500000,7.000000,15.467740,\Rx:=0.000000,\Ry:=4.827931),vel1,zoneval,Extruder\WObj:=Workobject_1;
MoveL RelTool (p1,60.000000,7.000000,14.360829,\Rx:=0.000000,\Ry:=5.885785),vel1,zoneval,Extruder\WObj:=Workobject_1;
MoveL RelTool (p1,62.500000,7.000000,12.917427,\Rx:=0.000000,\Ry:=8.074346),vel1,zoneval,Extruder\WObj:=Workobject_1;
MoveL RelTool (p1,65.000000,7.000000,10.805704,\Rx:=0.000000,\Ry:=10.911608),vel1,zoneval,Extruder\WObj:=Workobject_1;
MoveL RelTool (p1,67.500000,7.000000,8.322622,\Rx:=0.000000,\Ry:=4.473458),vel1,zoneval,Extruder\WObj:=Workobject_1;
MoveL RelTool (p1,70.000000,7.000000,8.000000,\Rx:=0.000000,\Ry:=-0.000000),vel1,zoneval,Extruder\WObj:=Workobject_1;
MoveL RelTool (p1,72.500000,7.000000,8.000000,\Rx:=0.000000,\Ry:=-0.000000),vel1,zoneval,Extruder\WObj:=Workobject_1;
MoveL RelTool (p1,75.000000,7.000000,8.000000,\Rx:=0.000000,\Ry:=-0.000000),vel1,zoneval,Extruder\WObj:=Workobject_1;
MoveL RelTool (p1,77.500000,7.000000,8.000000,\Rx:=0.000000,\Ry:=-0.000000),vel1,zoneval,Extruder\WObj:=Workobject_1;
MoveL RelTool (p1,80.000000,7.000000,8.000000,\Rx:=0.000000,\Ry:=-0.000000),vel1,zoneval,Extruder\WObj:=Workobject_1;
MoveL RelTool (p1,82.500000,7.000000,8.000000,\Rx:=0.000000,\Ry:=-0.000000),vel1,zoneval,Extruder\WObj:=Workobject_1;
MoveL RelTool (p1,80.500000,7.500000,8.000000,\Rx:=0.000000,\Ry:=0.000000),vel1,zoneval,Extruder\WObj:=Workobject_1;
MoveL RelTool (p1,78.000000,7.500000,8.000000,\Rx:=0.000000,\Ry:=0.000000),vel1,zoneval,Extruder\WObj:=Workobject_1;
MoveL RelTool (p1,75.500000,7.500000,8.000000,\Rx:=0.000000,\Ry:=0.000000),vel1,zoneval,Extruder\WObj:=Workobject_1;
MoveL RelTool (p1,73.000000,7.500000,8.000000,\Rx:=0.000000,\Ry:=0.000000),vel1,zoneval,Extruder\WObj:=Workobject_1;
MoveL RelTool (p1,70.500000,7.500000,8.000000,\Rx:=0.000000,\Ry:=0.000000),vel1,zoneval,Extruder\WObj:=Workobject_1;
MoveL RelTool (p1,68.000000,7.500000,8.139346,\Rx:=0.000000,\Ry:=4.473458),vel1,zoneval,Extruder\WObj:=Workobject_1;
MoveL RelTool (p1,65.500000,7.500000,10.229951,\Rx:=0.000000,\Ry:=10.902195),vel1,zoneval,Extruder\WObj:=Workobject_1;
MoveL RelTool (p1,63.000000,7.500000,12.550709,\Rx:=0.000000,\Ry:=8.053810),vel1,zoneval,Extruder\WObj:=Workobject_1;
MoveL RelTool (p1,60.500000,7.500000,14.111990,\Rx:=0.000000,\Ry:=5.885785),vel1,zoneval,Extruder\WObj:=Workobject_1;
MoveL RelTool (p1,58.000000,7.500000,15.269219,\Rx:=0.000000,\Ry:=4.827931),vel1,zoneval,Extruder\WObj:=Workobject_1;
MoveL RelTool (p1,55.500000,7.500000,16.163332,\Rx:=0.000000,\Ry:=3.853351),vel1,zoneval,Extruder\WObj:=Workobject_1;
MoveL RelTool (p1,53.000000,7.500000,16.838976,\Rx:=0.000000,\Ry:=2.916112),vel1,zoneval,Extruder\WObj:=Workobject_1;
MoveL RelTool (p1,50.500000,7.500000,17.351800,\Rx:=0.000000,\Ry:=2.025279),vel1,zoneval,Extruder\WObj:=Workobject_1;
MoveL RelTool (p1,48.000000,7.500000,17.710104,\Rx:=0.000000,\Ry:=1.180016),vel1,zoneval,Extruder\WObj:=Workobject_1;
MoveL RelTool (p1,45.500000,7.500000,17.924268,\Rx:=0.000000,\Ry:=0.518449),vel1,zoneval,Extruder\WObj:=Workobject_1;
MoveL RelTool (p1,43.000000,7.500000,17.996982,\Rx:=0.000000,\Ry:=-0.132553),vel1,zoneval,Extruder\WObj:=Workobject_1;
MoveL RelTool (p1,40.500000,7.500000,17.927163,\Rx:=0.000000,\Ry:=-0.544309),vel1,zoneval,Extruder\WObj:=Workobject_1;
MoveL RelTool (p1,38.000000,7.500000,17.721876,\Rx:=0.000000,\Ry:=-1.272729),vel1,zoneval,Extruder\WObj:=Workobject_1;
MoveL RelTool (p1,35.500000,7.500000,17.381188,\Rx:=0.000000,\Ry:=-2.131683),vel1,zoneval,Extruder\WObj:=Workobject_1;
MoveL RelTool (p1,33.000000,7.500000,16.880874,\Rx:=0.000000,\Ry:=-3.054804),vel1,zoneval,Extruder\WObj:=Workobject_1;
MoveL RelTool (p1,30.500000,7.500000,16.216792,\Rx:=0.000000,\Ry:=-4.018116),vel1,zoneval,Extruder\WObj:=Workobject_1;
MoveL RelTool (p1,28.000000,7.500000,15.334840,\Rx:=0.000000,\Ry:=-5.054525),vel1,zoneval,Extruder\WObj:=Workobject_1;
MoveL RelTool (p1,25.500000,7.500000,14.195301,\Rx:=0.000000,\Ry:=-6.198553),vel1,zoneval,Extruder\WObj:=Workobject_1;
MoveL RelTool (p1,23.000000,7.500000,12.678489,\Rx:=0.000000,\Ry:=-8.160407),vel1,zoneval,Extruder\WObj:=Workobject_1;
MoveL RelTool (p1,20.500000,7.500000,10.425592,\Rx:=0.000000,\Ry:=-11.197134),vel1,zoneval,Extruder\WObj:=Workobject_1;
MoveL RelTool (p1,18.000000,7.500000,8.180767,\Rx:=0.000000,\Ry:=-3.082616),vel1,zoneval,Extruder\WObj:=Workobject_1;
MoveL RelTool (p1,15.500000,7.500000,8.000000,\Rx:=0.000000,\Ry:=0.000000),vel1,zoneval,Extruder\WObj:=Workobject_1;
MoveL RelTool (p1,13.000000,7.500000,8.000000,\Rx:=0.000000,\Ry:=0.000000),vel1,zoneval,Extruder\WObj:=Workobject_1;
MoveL RelTool (p1,10.500000,7.500000,8.000000,\Rx:=0.000000,\Ry:=0.000000),vel1,zoneval,Extruder\WObj:=Workobject_1;
MoveL RelTool (p1,8.000000,7.500000,8.000000,\Rx:=0.000000,\Ry:=0.000000),vel1,zoneval,Extruder\WObj:=Workobject_1;
MoveL RelTool (p1,5.500000,7.500000,8.000000,\Rx:=0.000000,\Ry:=0.000000),vel1,zoneval,Extruder\WObj:=Workobject_1;
MoveL RelTool (p1,3.000000,7.500000,8.000000,\Rx:=0.000000,\Ry:=0.000000),vel1,zoneval,Extruder\WObj:=Workobject_1;
MoveL RelTool (p1,5.000000,8.000000,8.000000,\Rx:=0.000000,\Ry:=-0.000000),vel1,zoneval,Extruder\WObj:=Workobject_1;
MoveL RelTool (p1,7.500000,8.000000,8.000000,\Rx:=0.000000,\Ry:=-0.000000),vel1,zoneval,Extruder\WObj:=Workobject_1;
MoveL RelTool (p1,10.000000,8.000000,8.000000,\Rx:=0.000000,\Ry:=-0.000000),vel1,zoneval,Extruder\WObj:=Workobject_1;
MoveL RelTool (p1,12.500000,8.000000,8.000000,\Rx:=0.000000,\Ry:=-0.000000),vel1,zoneval,Extruder\WObj:=Workobject_1;
MoveL RelTool (p1,15.000000,8.000000,8.000000,\Rx:=0.000000,\Ry:=-0.000000),vel1,zoneval,Extruder\WObj:=Workobject_1;
MoveL RelTool (p1,17.500000,8.000000,8.057291,\Rx:=0.000000,\Ry:=-3.082616),vel1,zoneval,Extruder\WObj:=Workobject_1;
MoveL RelTool (p1,20.000000,8.000000,9.821760,\Rx:=0.000000,\Ry:=-11.198937),vel1,zoneval,Extruder\WObj:=Workobject_1;
MoveL RelTool (p1,22.500000,8.000000,12.306342,\Rx:=0.000000,\Ry:=-8.174155),vel1,zoneval,Extruder\WObj:=Workobject_1;
MoveL RelTool (p1,25.000000,8.000000,13.931837,\Rx:=0.000000,\Ry:=-6.198553),vel1,zoneval,Extruder\WObj:=Workobject_1;
MoveL RelTool (p1,27.500000,8.000000,15.125575,\Rx:=0.000000,\Ry:=-5.077061),vel1,zoneval,Extruder\WObj:=Workobject_1;
MoveL RelTool (p1,30.000000,8.000000,16.054193,\Rx:=0.000000,\Ry:=-4.018116),vel1,zoneval,Extruder\WObj:=Workobject_1;
MoveL RelTool (p1,32.500000,8.000000,16.758712,\Rx:=0.000000,\Ry:=-3.054804),vel1,zoneval,Extruder\WObj:=Workobject_1;
MoveL RelTool (p1,35.000000,8.000000,17.297700,\Rx:=0.000000,\Ry:=-2.131683),vel1,zoneval,Extruder\WObj:=Workobject_1;
MoveL RelTool (p1,37.500000,8.000000,17.672035,\Rx:=0.000000,\Ry:=-1.286021),vel1,zoneval,Extruder\WObj:=Workobject_1;
MoveL RelTool (p1,40.000000,8.000000,17.905452,\Rx:=0.000000,\Ry:=-0.572027),vel1,zoneval,Extruder\WObj:=Workobject_1;
MoveL RelTool (p1,42.500000,8.000000,17.992209,\Rx:=0.000000,\Ry:=-0.115153),vel1,zoneval,Extruder\WObj:=Workobject_1;
MoveL RelTool (p1,45.000000,8.000000,17.945442,\Rx:=0.000000,\Ry:=0.543320),vel1,zoneval,Extruder\WObj:=Workobject_1;
MoveL RelTool (p1,47.500000,8.000000,17.757402,\Rx:=0.000000,\Ry:=1.180016),vel1,zoneval,Extruder\WObj:=Workobject_1;
MoveL RelTool (p1,50.000000,8.000000,17.432501,\Rx:=0.000000,\Ry:=2.025279),vel1,zoneval,Extruder\WObj:=Workobject_1;
MoveL RelTool (p1,52.500000,8.000000,16.956476,\Rx:=0.000000,\Ry:=2.938011),vel1,zoneval,Extruder\WObj:=Workobject_1;
MoveL RelTool (p1,55.000000,8.000000,16.320430,\Rx:=0.000000,\Ry:=3.853351),vel1,zoneval,Extruder\WObj:=Workobject_1;
MoveL RelTool (p1,57.500000,8.000000,15.469165,\Rx:=0.000000,\Ry:=4.827931),vel1,zoneval,Extruder\WObj:=Workobject_1;
MoveL RelTool (p1,60.000000,8.000000,14.361428,\Rx:=0.000000,\Ry:=5.885785),vel1,zoneval,Extruder\WObj:=Workobject_1;
MoveL RelTool (p1,62.500000,8.000000,12.917010,\Rx:=0.000000,\Ry:=8.033226),vel1,zoneval,Extruder\WObj:=Workobject_1;
MoveL RelTool (p1,65.000000,8.000000,10.806997,\Rx:=0.000000,\Ry:=10.892765),vel1,zoneval,Extruder\WObj:=Workobject_1;
MoveL RelTool (p1,67.500000,8.000000,8.322622,\Rx:=0.000000,\Ry:=4.473458),vel1,zoneval,Extruder\WObj:=Workobject_1;
MoveL RelTool (p1,70.000000,8.000000,8.000000,\Rx:=0.000000,\Ry:=-0.000000),vel1,zoneval,Extruder\WObj:=Workobject_1;
MoveL RelTool (p1,72.500000,8.000000,8.000000,\Rx:=0.000000,\Ry:=-0.000000),vel1,zoneval,Extruder\WObj:=Workobject_1;
MoveL RelTool (p1,75.000000,8.000000,8.000000,\Rx:=0.000000,\Ry:=-0.000000),vel1,zoneval,Extruder\WObj:=Workobject_1;
MoveL RelTool (p1,77.500000,8.000000,8.000000,\Rx:=0.000000,\Ry:=-0.000000),vel1,zoneval,Extruder\WObj:=Workobject_1;
MoveL RelTool (p1,80.000000,8.000000,8.000000,\Rx:=0.000000,\Ry:=-0.000000),vel1,zoneval,Extruder\WObj:=Workobject_1;
MoveL RelTool (p1,82.500000,8.000000,8.000000,\Rx:=0.000000,\Ry:=-0.000000),vel1,zoneval,Extruder\WObj:=Workobject_1;
MoveL RelTool (p1,80.500000,8.500000,8.000000,\Rx:=0.000000,\Ry:=0.000000),vel1,zoneval,Extruder\WObj:=Workobject_1;
MoveL RelTool (p1,78.000000,8.500000,8.000000,\Rx:=0.000000,\Ry:=0.000000),vel1,zoneval,Extruder\WObj:=Workobject_1;
MoveL RelTool (p1,75.500000,8.500000,8.000000,\Rx:=0.000000,\Ry:=0.000000),vel1,zoneval,Extruder\WObj:=Workobject_1;
MoveL RelTool (p1,73.000000,8.500000,8.000000,\Rx:=0.000000,\Ry:=0.000000),vel1,zoneval,Extruder\WObj:=Workobject_1;
MoveL RelTool (p1,70.500000,8.500000,8.000000,\Rx:=0.000000,\Ry:=0.000000),vel1,zoneval,Extruder\WObj:=Workobject_1;
MoveL RelTool (p1,68.000000,8.500000,8.139346,\Rx:=0.000000,\Ry:=4.473458),vel1,zoneval,Extruder\WObj:=Workobject_1;
MoveL RelTool (p1,65.500000,8.500000,10.232968,\Rx:=0.000000,\Ry:=10.883320),vel1,zoneval,Extruder\WObj:=Workobject_1;
MoveL RelTool (p1,63.000000,8.500000,12.552774,\Rx:=0.000000,\Ry:=8.012593),vel1,zoneval,Extruder\WObj:=Workobject_1;
MoveL RelTool (p1,60.500000,8.500000,14.112588,\Rx:=0.000000,\Ry:=5.885785),vel1,zoneval,Extruder\WObj:=Workobject_1;
MoveL RelTool (p1,58.000000,8.500000,15.270644,\Rx:=0.000000,\Ry:=4.827931),vel1,zoneval,Extruder\WObj:=Workobject_1;
MoveL RelTool (p1,55.500000,8.500000,16.165295,\Rx:=0.000000,\Ry:=3.853351),vel1,zoneval,Extruder\WObj:=Workobject_1;
MoveL RelTool (p1,53.000000,8.500000,16.839041,\Rx:=0.000000,\Ry:=2.978510),vel1,zoneval,Extruder\WObj:=Workobject_1;
MoveL RelTool (p1,50.500000,8.500000,17.352782,\Rx:=0.000000,\Ry:=2.025279),vel1,zoneval,Extruder\WObj:=Workobject_1;
MoveL RelTool (p1,48.000000,8.500000,17.711755,\Rx:=0.000000,\Ry:=1.180016),vel1,zoneval,Extruder\WObj:=Workobject_1;
MoveL RelTool (p1,45.500000,8.500000,17.923917,\Rx:=0.000000,\Ry:=0.568186),vel1,zoneval,Extruder\WObj:=Workobject_1;
MoveL RelTool (p1,43.000000,8.500000,17.996480,\Rx:=0.000000,\Ry:=-0.097752),vel1,zoneval,Extruder\WObj:=Workobject_1;
MoveL RelTool (p1,40.500000,8.500000,17.928699,\Rx:=0.000000,\Ry:=-0.599740),vel1,zoneval,Extruder\WObj:=Workobject_1;
MoveL RelTool (p1,38.000000,8.500000,17.723544,\Rx:=0.000000,\Ry:=-1.299310),vel1,zoneval,Extruder\WObj:=Workobject_1;
MoveL RelTool (p1,35.500000,8.500000,17.383216,\Rx:=0.000000,\Ry:=-2.131683),vel1,zoneval,Extruder\WObj:=Workobject_1;
MoveL RelTool (p1,33.000000,8.500000,16.881186,\Rx:=0.000000,\Ry:=-3.054804),vel1,zoneval,Extruder\WObj:=Workobject_1;
MoveL RelTool (p1,30.500000,8.500000,16.218086,\Rx:=0.000000,\Ry:=-4.018116),vel1,zoneval,Extruder\WObj:=Workobject_1;
MoveL RelTool (p1,28.000000,8.500000,15.337633,\Rx:=0.000000,\Ry:=-5.099563),vel1,zoneval,Extruder\WObj:=Workobject_1;
MoveL RelTool (p1,25.500000,8.500000,14.197701,\Rx:=0.000000,\Ry:=-6.198553),vel1,zoneval,Extruder\WObj:=Workobject_1;
MoveL RelTool (p1,23.000000,8.500000,12.681847,\Rx:=0.000000,\Ry:=-8.187882),vel1,zoneval,Extruder\WObj:=Workobject_1;
MoveL RelTool (p1,20.500000,8.500000,10.426515,\Rx:=0.000000,\Ry:=-11.200739),vel1,zoneval,Extruder\WObj:=Workobject_1;
MoveL RelTool (p1,18.000000,8.500000,8.180767,\Rx:=0.000000,\Ry:=-3.082616),vel1,zoneval,Extruder\WObj:=Workobject_1;
MoveL RelTool (p1,15.500000,8.500000,8.000000,\Rx:=0.000000,\Ry:=0.000000),vel1,zoneval,Extruder\WObj:=Workobject_1;
MoveL RelTool (p1,13.000000,8.500000,8.000000,\Rx:=0.000000,\Ry:=0.000000),vel1,zoneval,Extruder\WObj:=Workobject_1;
MoveL RelTool (p1,10.500000,8.500000,8.000000,\Rx:=0.000000,\Ry:=0.000000),vel1,zoneval,Extruder\WObj:=Workobject_1;
MoveL RelTool (p1,8.000000,8.500000,8.000000,\Rx:=0.000000,\Ry:=0.000000),vel1,zoneval,Extruder\WObj:=Workobject_1;
MoveL RelTool (p1,5.500000,8.500000,8.000000,\Rx:=0.000000,\Ry:=0.000000),vel1,zoneval,Extruder\WObj:=Workobject_1;
MoveL RelTool (p1,3.000000,8.500000,8.000000,\Rx:=0.000000,\Ry:=0.000000),vel1,zoneval,Extruder\WObj:=Workobject_1;
MoveL RelTool (p1,5.000000,9.000000,8.000000,\Rx:=0.000000,\Ry:=-0.000000),vel1,zoneval,Extruder\WObj:=Workobject_1;
MoveL RelTool (p1,7.500000,9.000000,8.000000,\Rx:=0.000000,\Ry:=-0.000000),vel1,zoneval,Extruder\WObj:=Workobject_1;
MoveL RelTool (p1,10.000000,9.000000,8.000000,\Rx:=0.000000,\Ry:=-0.000000),vel1,zoneval,Extruder\WObj:=Workobject_1;
MoveL RelTool (p1,12.500000,9.000000,8.000000,\Rx:=0.000000,\Ry:=-0.000000),vel1,zoneval,Extruder\WObj:=Workobject_1;
MoveL RelTool (p1,15.000000,9.000000,8.000000,\Rx:=0.000000,\Ry:=-0.000000),vel1,zoneval,Extruder\WObj:=Workobject_1;
MoveL RelTool (p1,17.500000,9.000000,8.057291,\Rx:=0.000000,\Ry:=-3.082616),vel1,zoneval,Extruder\WObj:=Workobject_1;
MoveL RelTool (p1,20.000000,9.000000,9.822334,\Rx:=0.000000,\Ry:=-11.202541),vel1,zoneval,Extruder\WObj:=Workobject_1;
MoveL RelTool (p1,22.500000,9.000000,12.308018,\Rx:=0.000000,\Ry:=-8.201245),vel1,zoneval,Extruder\WObj:=Workobject_1;
MoveL RelTool (p1,25.000000,9.000000,13.934237,\Rx:=0.000000,\Ry:=-6.198553),vel1,zoneval,Extruder\WObj:=Workobject_1;
MoveL RelTool (p1,27.500000,9.000000,15.126285,\Rx:=0.000000,\Ry:=-5.122032),vel1,zoneval,Extruder\WObj:=Workobject_1;
MoveL RelTool (p1,30.000000,9.000000,16.055487,\Rx:=0.000000,\Ry:=-4.018116),vel1,zoneval,Extruder\WObj:=Workobject_1;
MoveL RelTool (p1,32.500000,9.000000,16.759024,\Rx:=0.000000,\Ry:=-3.054804),vel1,zoneval,Extruder\WObj:=Workobject_1;
MoveL RelTool (p1,35.000000,9.000000,17.299727,\Rx:=0.000000,\Ry:=-2.131683),vel1,zoneval,Extruder\WObj:=Workobject_1;
MoveL RelTool (p1,37.500000,9.000000,17.672649,\Rx:=0.000000,\Ry:=-1.312597),vel1,zoneval,Extruder\WObj:=Workobject_1;
MoveL RelTool (p1,40.000000,9.000000,17.904806,\Rx:=0.000000,\Ry:=-0.627447),vel1,zoneval,Extruder\WObj:=Workobject_1;
MoveL RelTool (p1,42.500000,9.000000,17.993073,\Rx:=0.000000,\Ry:=-0.080351),vel1,zoneval,Extruder\WObj:=Workobject_1;
MoveL RelTool (p1,45.000000,9.000000,17.947048,\Rx:=0.000000,\Ry:=0.593049),vel1,zoneval,Extruder\WObj:=Workobject_1;
MoveL RelTool (p1,47.500000,9.000000,17.759053,\Rx:=0.000000,\Ry:=1.180016),vel1,zoneval,Extruder\WObj:=Workobject_1;
MoveL RelTool (p1,50.000000,9.000000,17.433483,\Rx:=0.000000,\Ry:=2.025279),vel1,zoneval,Extruder\WObj:=Workobject_1;
MoveL RelTool (p1,52.500000,9.000000,16.959901,\Rx:=0.000000,\Ry:=3.018948),vel1,zoneval,Extruder\WObj:=Workobject_1;
MoveL RelTool (p1,55.000000,9.000000,16.322393,\Rx:=0.000000,\Ry:=3.853351),vel1,zoneval,Extruder\WObj:=Workobject_1;
MoveL RelTool (p1,57.500000,9.000000,15.470591,\Rx:=0.000000,\Ry:=4.827931),vel1,zoneval,Extruder\WObj:=Workobject_1;
MoveL RelTool (p1,60.000000,9.000000,14.362026,\Rx:=0.000000,\Ry:=5.885785),vel1,zoneval,Extruder\WObj:=Workobject_1;
MoveL RelTool (p1,62.500000,9.000000,12.916593,\Rx:=0.000000,\Ry:=8.000776),vel1,zoneval,Extruder\WObj:=Workobject_1;
MoveL RelTool (p1,65.000000,9.000000,10.808291,\Rx:=0.000000,\Ry:=10.873858),vel1,zoneval,Extruder\WObj:=Workobject_1;
MoveL RelTool (p1,67.500000,9.000000,8.322622,\Rx:=0.000000,\Ry:=4.473458),vel1,zoneval,Extruder\WObj:=Workobject_1;
MoveL RelTool (p1,70.000000,9.000000,8.000000,\Rx:=0.000000,\Ry:=-0.000000),vel1,zoneval,Extruder\WObj:=Workobject_1;
MoveL RelTool (p1,72.500000,9.000000,8.000000,\Rx:=0.000000,\Ry:=-0.000000),vel1,zoneval,Extruder\WObj:=Workobject_1;
MoveL RelTool (p1,75.000000,9.000000,8.000000,\Rx:=0.000000,\Ry:=-0.000000),vel1,zoneval,Extruder\WObj:=Workobject_1;
MoveL RelTool (p1,77.500000,9.000000,8.000000,\Rx:=0.000000,\Ry:=-0.000000),vel1,zoneval,Extruder\WObj:=Workobject_1;
MoveL RelTool (p1,80.000000,9.000000,8.000000,\Rx:=0.000000,\Ry:=-0.000000),vel1,zoneval,Extruder\WObj:=Workobject_1;
MoveL RelTool (p1,82.500000,9.000000,8.000000,\Rx:=0.000000,\Ry:=-0.000000),vel1,zoneval,Extruder\WObj:=Workobject_1;
MoveL RelTool (p1,80.500000,9.500000,8.000000,\Rx:=0.000000,\Ry:=0.000000),vel1,zoneval,Extruder\WObj:=Workobject_1;
MoveL RelTool (p1,78.000000,9.500000,8.000000,\Rx:=0.000000,\Ry:=0.000000),vel1,zoneval,Extruder\WObj:=Workobject_1;
MoveL RelTool (p1,75.500000,9.500000,8.000000,\Rx:=0.000000,\Ry:=0.000000),vel1,zoneval,Extruder\WObj:=Workobject_1;
MoveL RelTool (p1,73.000000,9.500000,8.000000,\Rx:=0.000000,\Ry:=0.000000),vel1,zoneval,Extruder\WObj:=Workobject_1;
MoveL RelTool (p1,70.500000,9.500000,8.000000,\Rx:=0.000000,\Ry:=0.000000),vel1,zoneval,Extruder\WObj:=Workobject_1;
MoveL RelTool (p1,68.000000,9.500000,8.139346,\Rx:=0.000000,\Ry:=4.473458),vel1,zoneval,Extruder\WObj:=Workobject_1;
MoveL RelTool (p1,65.500000,9.500000,10.235985,\Rx:=0.000000,\Ry:=10.864380),vel1,zoneval,Extruder\WObj:=Workobject_1;
MoveL RelTool (p1,63.000000,9.500000,12.553580,\Rx:=0.000000,\Ry:=7.992204),vel1,zoneval,Extruder\WObj:=Workobject_1;
MoveL RelTool (p1,60.500000,9.500000,14.113187,\Rx:=0.000000,\Ry:=5.885785),vel1,zoneval,Extruder\WObj:=Workobject_1;
MoveL RelTool (p1,58.000000,9.500000,15.272070,\Rx:=0.000000,\Ry:=4.823420),vel1,zoneval,Extruder\WObj:=Workobject_1;
MoveL RelTool (p1,55.500000,9.500000,16.167258,\Rx:=0.000000,\Ry:=3.853351),vel1,zoneval,Extruder\WObj:=Workobject_1;
MoveL RelTool (p1,53.000000,9.500000,16.839107,\Rx:=0.000000,\Ry:=3.059324),vel1,zoneval,Extruder\WObj:=Workobject_1;
MoveL RelTool (p1,50.500000,9.500000,17.353763,\Rx:=0.000000,\Ry:=2.025279),vel1,zoneval,Extruder\WObj:=Workobject_1;
MoveL RelTool (p1,48.000000,9.500000,17.713407,\Rx:=0.000000,\Ry:=1.180016),vel1,zoneval,Extruder\WObj:=Workobject_1;
MoveL RelTool (p1,45.500000,9.500000,17.923567,\Rx:=0.000000,\Ry:=0.600766),vel1,zoneval,Extruder\WObj:=Workobject_1;
MoveL RelTool (p1,43.000000,9.500000,17.995977,\Rx:=0.000000,\Ry:=-0.062950),vel1,zoneval,Extruder\WObj:=Workobject_1;
MoveL RelTool (p1,40.500000,9.500000,17.930234,\Rx:=0.000000,\Ry:=-0.655148),vel1,zoneval,Extruder\WObj:=Workobject_1;
MoveL RelTool (p1,38.000000,9.500000,17.725211,\Rx:=0.000000,\Ry:=-1.325880),vel1,zoneval,Extruder\WObj:=Workobject_1;
MoveL RelTool (p1,35.500000,9.500000,17.385243,\Rx:=0.000000,\Ry:=-2.131683),vel1,zoneval,Extruder\WObj:=Workobject_1;
MoveL RelTool (p1,33.000000,9.500000,16.881497,\Rx:=0.000000,\Ry:=-3.051292),vel1,zoneval,Extruder\WObj:=Workobject_1;
MoveL RelTool (p1,30.500000,9.500000,16.219380,\Rx:=0.000000,\Ry:=-4.018116),vel1,zoneval,Extruder\WObj:=Workobject_1;
MoveL RelTool (p1,28.000000,9.500000,15.340425,\Rx:=0.000000,\Ry:=-5.144467),vel1,zoneval,Extruder\WObj:=Workobject_1;
MoveL RelTool (p1,25.500000,9.500000,14.200100,\Rx:=0.000000,\Ry:=-6.198553),vel1,zoneval,Extruder\WObj:=Workobject_1;
MoveL RelTool (p1,23.000000,9.500000,12.683149,\Rx:=0.000000,\Ry:=-8.181774),vel1,zoneval,Extruder\WObj:=Workobject_1;
MoveL RelTool (p1,20.500000,9.500000,10.427438,\Rx:=0.000000,\Ry:=-11.204342),vel1,zoneval,Extruder\WObj:=Workobject_1;
MoveL RelTool (p1,18.000000,9.500000,8.180767,\Rx:=0.000000,\Ry:=-3.082616),vel1,zoneval,Extruder\WObj:=Workobject_1;
MoveL RelTool (p1,15.500000,9.500000,8.000000,\Rx:=0.000000,\Ry:=0.000000),vel1,zoneval,Extruder\WObj:=Workobject_1;
MoveL RelTool (p1,13.000000,9.500000,8.000000,\Rx:=0.000000,\Ry:=0.000000),vel1,zoneval,Extruder\WObj:=Workobject_1;
MoveL RelTool (p1,10.500000,9.500000,8.000000,\Rx:=0.000000,\Ry:=0.000000),vel1,zoneval,Extruder\WObj:=Workobject_1;
MoveL RelTool (p1,8.000000,9.500000,8.000000,\Rx:=0.000000,\Ry:=0.000000),vel1,zoneval,Extruder\WObj:=Workobject_1;
MoveL RelTool (p1,5.500000,9.500000,8.000000,\Rx:=0.000000,\Ry:=0.000000),vel1,zoneval,Extruder\WObj:=Workobject_1;
MoveL RelTool (p1,3.000000,9.500000,8.000000,\Rx:=0.000000,\Ry:=0.000000),vel1,zoneval,Extruder\WObj:=Workobject_1;
MoveL RelTool (p1,5.000000,10.000000,8.000000,\Rx:=0.000000,\Ry:=-0.000000),vel1,zoneval,Extruder\WObj:=Workobject_1;
MoveL RelTool (p1,7.500000,10.000000,8.000000,\Rx:=0.000000,\Ry:=-0.000000),vel1,zoneval,Extruder\WObj:=Workobject_1;
MoveL RelTool (p1,10.000000,10.000000,8.000000,\Rx:=0.000000,\Ry:=-0.000000),vel1,zoneval,Extruder\WObj:=Workobject_1;
MoveL RelTool (p1,12.500000,10.000000,8.000000,\Rx:=0.000000,\Ry:=-0.000000),vel1,zoneval,Extruder\WObj:=Workobject_1;
MoveL RelTool (p1,15.000000,10.000000,8.000000,\Rx:=0.000000,\Ry:=-0.000000),vel1,zoneval,Extruder\WObj:=Workobject_1;
MoveL RelTool (p1,17.500000,10.000000,8.057291,\Rx:=0.000000,\Ry:=-3.082616),vel1,zoneval,Extruder\WObj:=Workobject_1;
MoveL RelTool (p1,20.000000,10.000000,9.822909,\Rx:=0.000000,\Ry:=-11.206143),vel1,zoneval,Extruder\WObj:=Workobject_1;
MoveL RelTool (p1,22.500000,10.000000,12.309694,\Rx:=0.000000,\Ry:=-8.162259),vel1,zoneval,Extruder\WObj:=Workobject_1;
MoveL RelTool (p1,25.000000,10.000000,13.936636,\Rx:=0.000000,\Ry:=-6.198553),vel1,zoneval,Extruder\WObj:=Workobject_1;
MoveL RelTool (p1,27.500000,10.000000,15.126996,\Rx:=0.000000,\Ry:=-5.166868),vel1,zoneval,Extruder\WObj:=Workobject_1;
MoveL RelTool (p1,30.000000,10.000000,16.056781,\Rx:=0.000000,\Ry:=-4.018116),vel1,zoneval,Extruder\WObj:=Workobject_1;
MoveL RelTool (p1,32.500000,10.000000,16.760896,\Rx:=0.000000,\Ry:=-3.017271),vel1,zoneval,Extruder\WObj:=Workobject_1;
MoveL RelTool (p1,35.000000,10.000000,17.301755,\Rx:=0.000000,\Ry:=-2.131683),vel1,zoneval,Extruder\WObj:=Workobject_1;
MoveL RelTool (p1,37.500000,10.000000,17.673262,\Rx:=0.000000,\Ry:=-1.339161),vel1,zoneval,Extruder\WObj:=Workobject_1;
MoveL RelTool (p1,40.000000,10.000000,17.904160,\Rx:=0.000000,\Ry:=-0.682843),vel1,zoneval,Extruder\WObj:=Workobject_1;
MoveL RelTool (p1,42.500000,10.000000,17.993937,\Rx:=0.000000,\Ry:=-0.045548),vel1,zoneval,Extruder\WObj:=Workobject_1;
MoveL RelTool (p1,45.000000,10.000000,17.947001,\Rx:=0.000000,\Ry:=0.600766),vel1,zoneval,Extruder\WObj:=Workobject_1;
MoveL RelTool (p1,47.500000,10.000000,17.760705,\Rx:=0.000000,\Ry:=1.180016),vel1,zoneval,Extruder\WObj:=Workobject_1;
MoveL RelTool (p1,50.000000,10.000000,17.434464,\Rx:=0.000000,\Ry:=2.025279),vel1,zoneval,Extruder\WObj:=Workobject_1;
MoveL RelTool (p1,52.500000,10.000000,16.963326,\Rx:=0.000000,\Ry:=3.099637),vel1,zoneval,Extruder\WObj:=Workobject_1;
MoveL RelTool (p1,55.000000,10.000000,16.324242,\Rx:=0.000000,\Ry:=3.850713),vel1,zoneval,Extruder\WObj:=Workobject_1;
MoveL RelTool (p1,57.500000,10.000000,15.471596,\Rx:=0.000000,\Ry:=4.818681),vel1,zoneval,Extruder\WObj:=Workobject_1;
MoveL RelTool (p1,60.000000,10.000000,14.362625,\Rx:=0.000000,\Ry:=5.885785),vel1,zoneval,Extruder\WObj:=Workobject_1;
MoveL RelTool (p1,62.500000,10.000000,12.916175,\Rx:=0.000000,\Ry:=7.983623),vel1,zoneval,Extruder\WObj:=Workobject_1;
MoveL RelTool (p1,65.000000,10.000000,10.809584,\Rx:=0.000000,\Ry:=10.854886),vel1,zoneval,Extruder\WObj:=Workobject_1;
MoveL RelTool (p1,67.500000,10.000000,8.322622,\Rx:=0.000000,\Ry:=4.473458),vel1,zoneval,Extruder\WObj:=Workobject_1;
MoveL RelTool (p1,70.000000,10.000000,8.000000,\Rx:=0.000000,\Ry:=-0.000000),vel1,zoneval,Extruder\WObj:=Workobject_1;
MoveL RelTool (p1,72.500000,10.000000,8.000000,\Rx:=0.000000,\Ry:=-0.000000),vel1,zoneval,Extruder\WObj:=Workobject_1;
MoveL RelTool (p1,75.000000,10.000000,8.000000,\Rx:=0.000000,\Ry:=-0.000000),vel1,zoneval,Extruder\WObj:=Workobject_1;
MoveL RelTool (p1,77.500000,10.000000,8.000000,\Rx:=0.000000,\Ry:=-0.000000),vel1,zoneval,Extruder\WObj:=Workobject_1;
MoveL RelTool (p1,80.000000,10.000000,8.000000,\Rx:=0.000000,\Ry:=-0.000000),vel1,zoneval,Extruder\WObj:=Workobject_1;
MoveL RelTool (p1,82.500000,10.000000,8.000000,\Rx:=0.000000,\Ry:=-0.000000),vel1,zoneval,Extruder\WObj:=Workobject_1;
MoveL RelTool (p1,80.500000,10.500000,8.000000,\Rx:=0.000000,\Ry:=0.000000),vel1,zoneval,Extruder\WObj:=Workobject_1;
MoveL RelTool (p1,78.000000,10.500000,8.000000,\Rx:=0.000000,\Ry:=0.000000),vel1,zoneval,Extruder\WObj:=Workobject_1;
MoveL RelTool (p1,75.500000,10.500000,8.000000,\Rx:=0.000000,\Ry:=0.000000),vel1,zoneval,Extruder\WObj:=Workobject_1;
MoveL RelTool (p1,73.000000,10.500000,8.000000,\Rx:=0.000000,\Ry:=0.000000),vel1,zoneval,Extruder\WObj:=Workobject_1;
MoveL RelTool (p1,70.500000,10.500000,8.000000,\Rx:=0.000000,\Ry:=0.000000),vel1,zoneval,Extruder\WObj:=Workobject_1;
MoveL RelTool (p1,68.000000,10.500000,8.139346,\Rx:=0.000000,\Ry:=4.473458),vel1,zoneval,Extruder\WObj:=Workobject_1;
MoveL RelTool (p1,65.500000,10.500000,10.239002,\Rx:=0.000000,\Ry:=10.845376),vel1,zoneval,Extruder\WObj:=Workobject_1;
MoveL RelTool (p1,63.000000,10.500000,12.554191,\Rx:=0.000000,\Ry:=7.975033),vel1,zoneval,Extruder\WObj:=Workobject_1;
MoveL RelTool (p1,60.500000,10.500000,14.113786,\Rx:=0.000000,\Ry:=5.885785),vel1,zoneval,Extruder\WObj:=Workobject_1;
MoveL RelTool (p1,58.000000,10.500000,15.273495,\Rx:=0.000000,\Ry:=4.813941),vel1,zoneval,Extruder\WObj:=Workobject_1;
MoveL RelTool (p1,55.500000,10.500000,16.169221,\Rx:=0.000000,\Ry:=3.828481),vel1,zoneval,Extruder\WObj:=Workobject_1;
MoveL RelTool (p1,53.000000,10.500000,16.840378,\Rx:=0.000000,\Ry:=3.111016),vel1,zoneval,Extruder\WObj:=Workobject_1;
MoveL RelTool (p1,50.500000,10.500000,17.354744,\Rx:=0.000000,\Ry:=2.032422),vel1,zoneval,Extruder\WObj:=Workobject_1;
MoveL RelTool (p1,48.000000,10.500000,17.715058,\Rx:=0.000000,\Ry:=1.180016),vel1,zoneval,Extruder\WObj:=Workobject_1;
MoveL RelTool (p1,45.500000,10.500000,17.923216,\Rx:=0.000000,\Ry:=0.600766),vel1,zoneval,Extruder\WObj:=Workobject_1;
MoveL RelTool (p1,43.000000,10.500000,17.995475,\Rx:=0.000000,\Ry:=-0.028146),vel1,zoneval,Extruder\WObj:=Workobject_1;
MoveL RelTool (p1,40.500000,10.500000,17.931769,\Rx:=0.000000,\Ry:=-0.710531),vel1,zoneval,Extruder\WObj:=Workobject_1;
MoveL RelTool (p1,38.000000,10.500000,17.726603,\Rx:=0.000000,\Ry:=-1.345493),vel1,zoneval,Extruder\WObj:=Workobject_1;
MoveL RelTool (p1,35.500000,10.500000,17.387270,\Rx:=0.000000,\Ry:=-2.131683),vel1,zoneval,Extruder\WObj:=Workobject_1;
MoveL RelTool (p1,33.000000,10.500000,16.881809,\Rx:=0.000000,\Ry:=-2.983205),vel1,zoneval,Extruder\WObj:=Workobject_1;
MoveL RelTool (p1,30.500000,10.500000,16.220675,\Rx:=0.000000,\Ry:=-4.018116),vel1,zoneval,Extruder\WObj:=Workobject_1;
MoveL RelTool (p1,28.000000,10.500000,15.343218,\Rx:=0.000000,\Ry:=-5.184167),vel1,zoneval,Extruder\WObj:=Workobject_1;
MoveL RelTool (p1,25.500000,10.500000,14.202499,\Rx:=0.000000,\Ry:=-6.198553),vel1,zoneval,Extruder\WObj:=Workobject_1;
MoveL RelTool (p1,23.000000,10.500000,12.682436,\Rx:=0.000000,\Ry:=-8.142699),vel1,zoneval,Extruder\WObj:=Workobject_1;
MoveL RelTool (p1,20.500000,10.500000,10.428360,\Rx:=0.000000,\Ry:=-11.207942),vel1,zoneval,Extruder\WObj:=Workobject_1;
MoveL RelTool (p1,18.000000,10.500000,8.180767,\Rx:=0.000000,\Ry:=-3.082616),vel1,zoneval,Extruder\WObj:=Workobject_1;
MoveL RelTool (p1,15.500000,10.500000,8.000000,\Rx:=0.000000,\Ry:=0.000000),vel1,zoneval,Extruder\WObj:=Workobject_1;
MoveL RelTool (p1,13.000000,10.500000,8.000000,\Rx:=0.000000,\Ry:=0.000000),vel1,zoneval,Extruder\WObj:=Workobject_1;
MoveL RelTool (p1,10.500000,10.500000,8.000000,\Rx:=0.000000,\Ry:=0.000000),vel1,zoneval,Extruder\WObj:=Workobject_1;
MoveL RelTool (p1,8.000000,10.500000,8.000000,\Rx:=0.000000,\Ry:=0.000000),vel1,zoneval,Extruder\WObj:=Workobject_1;
MoveL RelTool (p1,5.500000,10.500000,8.000000,\Rx:=0.000000,\Ry:=0.000000),vel1,zoneval,Extruder\WObj:=Workobject_1;
MoveL RelTool (p1,3.000000,10.500000,8.000000,\Rx:=0.000000,\Ry:=0.000000),vel1,zoneval,Extruder\WObj:=Workobject_1;
MoveL RelTool (p1,5.000000,11.000000,8.000000,\Rx:=0.000000,\Ry:=-0.000000),vel1,zoneval,Extruder\WObj:=Workobject_1;
MoveL RelTool (p1,7.500000,11.000000,8.000000,\Rx:=0.000000,\Ry:=-0.000000),vel1,zoneval,Extruder\WObj:=Workobject_1;
MoveL RelTool (p1,10.000000,11.000000,8.000000,\Rx:=0.000000,\Ry:=-0.000000),vel1,zoneval,Extruder\WObj:=Workobject_1;
MoveL RelTool (p1,12.500000,11.000000,8.000000,\Rx:=0.000000,\Ry:=-0.000000),vel1,zoneval,Extruder\WObj:=Workobject_1;
MoveL RelTool (p1,15.000000,11.000000,8.000000,\Rx:=0.000000,\Ry:=-0.000000),vel1,zoneval,Extruder\WObj:=Workobject_1;
MoveL RelTool (p1,17.500000,11.000000,8.057291,\Rx:=0.000000,\Ry:=-3.082616),vel1,zoneval,Extruder\WObj:=Workobject_1;
MoveL RelTool (p1,20.000000,11.000000,9.823483,\Rx:=0.000000,\Ry:=-11.209742),vel1,zoneval,Extruder\WObj:=Workobject_1;
MoveL RelTool (p1,22.500000,11.000000,12.311370,\Rx:=0.000000,\Ry:=-8.123094),vel1,zoneval,Extruder\WObj:=Workobject_1;
MoveL RelTool (p1,25.000000,11.000000,13.938364,\Rx:=0.000000,\Ry:=-6.211892),vel1,zoneval,Extruder\WObj:=Workobject_1;
MoveL RelTool (p1,27.500000,11.000000,15.128983,\Rx:=0.000000,\Ry:=-5.184167),vel1,zoneval,Extruder\WObj:=Workobject_1;
MoveL RelTool (p1,30.000000,11.000000,16.058075,\Rx:=0.000000,\Ry:=-4.018116),vel1,zoneval,Extruder\WObj:=Workobject_1;
MoveL RelTool (p1,32.500000,11.000000,16.764037,\Rx:=0.000000,\Ry:=-2.949096),vel1,zoneval,Extruder\WObj:=Workobject_1;
MoveL RelTool (p1,35.000000,11.000000,17.303782,\Rx:=0.000000,\Ry:=-2.131683),vel1,zoneval,Extruder\WObj:=Workobject_1;
MoveL RelTool (p1,37.500000,11.000000,17.673875,\Rx:=0.000000,\Ry:=-1.345493),vel1,zoneval,Extruder\WObj:=Workobject_1;
MoveL RelTool (p1,40.000000,11.000000,17.903514,\Rx:=0.000000,\Ry:=-0.738213),vel1,zoneval,Extruder\WObj:=Workobject_1;
MoveL RelTool (p1,42.500000,11.000000,17.994801,\Rx:=0.000000,\Ry:=-0.010745),vel1,zoneval,Extruder\WObj:=Workobject_1;
MoveL RelTool (p1,45.000000,11.000000,17.946650,\Rx:=0.000000,\Ry:=0.600766),vel1,zoneval,Extruder\WObj:=Workobject_1;
MoveL RelTool (p1,47.500000,11.000000,17.762356,\Rx:=0.000000,\Ry:=1.180016),vel1,zoneval,Extruder\WObj:=Workobject_1;
MoveL RelTool (p1,50.000000,11.000000,17.436096,\Rx:=0.000000,\Ry:=2.041421),vel1,zoneval,Extruder\WObj:=Workobject_1;
MoveL RelTool (p1,52.500000,11.000000,16.966751,\Rx:=0.000000,\Ry:=3.111016),vel1,zoneval,Extruder\WObj:=Workobject_1;
MoveL RelTool (p1,55.000000,11.000000,16.324290,\Rx:=0.000000,\Ry:=3.806226),vel1,zoneval,Extruder\WObj:=Workobject_1;
MoveL RelTool (p1,57.500000,11.000000,15.472590,\Rx:=0.000000,\Ry:=4.809200),vel1,zoneval,Extruder\WObj:=Workobject_1;
MoveL RelTool (p1,60.000000,11.000000,14.363836,\Rx:=0.000000,\Ry:=5.898266),vel1,zoneval,Extruder\WObj:=Workobject_1;
MoveL RelTool (p1,62.500000,11.000000,12.915758,\Rx:=0.000000,\Ry:=7.966435),vel1,zoneval,Extruder\WObj:=Workobject_1;
MoveL RelTool (p1,65.000000,11.000000,10.810878,\Rx:=0.000000,\Ry:=10.835850),vel1,zoneval,Extruder\WObj:=Workobject_1;
MoveL RelTool (p1,67.500000,11.000000,8.322622,\Rx:=0.000000,\Ry:=4.473458),vel1,zoneval,Extruder\WObj:=Workobject_1;
MoveL RelTool (p1,70.000000,11.000000,8.000000,\Rx:=0.000000,\Ry:=-0.000000),vel1,zoneval,Extruder\WObj:=Workobject_1;
MoveL RelTool (p1,72.500000,11.000000,8.000000,\Rx:=0.000000,\Ry:=-0.000000),vel1,zoneval,Extruder\WObj:=Workobject_1;
MoveL RelTool (p1,75.000000,11.000000,8.000000,\Rx:=0.000000,\Ry:=-0.000000),vel1,zoneval,Extruder\WObj:=Workobject_1;
MoveL RelTool (p1,77.500000,11.000000,8.000000,\Rx:=0.000000,\Ry:=-0.000000),vel1,zoneval,Extruder\WObj:=Workobject_1;
MoveL RelTool (p1,80.000000,11.000000,8.000000,\Rx:=0.000000,\Ry:=-0.000000),vel1,zoneval,Extruder\WObj:=Workobject_1;
MoveL RelTool (p1,82.500000,11.000000,8.000000,\Rx:=0.000000,\Ry:=-0.000000),vel1,zoneval,Extruder\WObj:=Workobject_1;
MoveL RelTool (p1,80.500000,11.500000,8.000000,\Rx:=0.000000,\Ry:=0.000000),vel1,zoneval,Extruder\WObj:=Workobject_1;
MoveL RelTool (p1,78.000000,11.500000,8.000000,\Rx:=0.000000,\Ry:=0.000000),vel1,zoneval,Extruder\WObj:=Workobject_1;
MoveL RelTool (p1,75.500000,11.500000,8.000000,\Rx:=0.000000,\Ry:=0.000000),vel1,zoneval,Extruder\WObj:=Workobject_1;
MoveL RelTool (p1,73.000000,11.500000,8.000000,\Rx:=0.000000,\Ry:=0.000000),vel1,zoneval,Extruder\WObj:=Workobject_1;
MoveL RelTool (p1,70.500000,11.500000,8.000000,\Rx:=0.000000,\Ry:=0.000000),vel1,zoneval,Extruder\WObj:=Workobject_1;
MoveL RelTool (p1,68.000000,11.500000,8.139346,\Rx:=0.000000,\Ry:=4.473458),vel1,zoneval,Extruder\WObj:=Workobject_1;
MoveL RelTool (p1,65.500000,11.500000,10.242019,\Rx:=0.000000,\Ry:=10.826307),vel1,zoneval,Extruder\WObj:=Workobject_1;
MoveL RelTool (p1,63.000000,11.500000,12.554802,\Rx:=0.000000,\Ry:=7.957829),vel1,zoneval,Extruder\WObj:=Workobject_1;
MoveL RelTool (p1,60.500000,11.500000,14.114384,\Rx:=0.000000,\Ry:=5.919672),vel1,zoneval,Extruder\WObj:=Workobject_1;
MoveL RelTool (p1,58.000000,11.500000,15.274921,\Rx:=0.000000,\Ry:=4.804458),vel1,zoneval,Extruder\WObj:=Workobject_1;
MoveL RelTool (p1,55.500000,11.500000,16.171184,\Rx:=0.000000,\Ry:=3.783947),vel1,zoneval,Extruder\WObj:=Workobject_1;
MoveL RelTool (p1,53.000000,11.500000,16.843803,\Rx:=0.000000,\Ry:=3.111016),vel1,zoneval,Extruder\WObj:=Workobject_1;
MoveL RelTool (p1,50.500000,11.500000,17.355726,\Rx:=0.000000,\Ry:=2.050418),vel1,zoneval,Extruder\WObj:=Workobject_1;
MoveL RelTool (p1,48.000000,11.500000,17.716710,\Rx:=0.000000,\Ry:=1.180016),vel1,zoneval,Extruder\WObj:=Workobject_1;
MoveL RelTool (p1,45.500000,11.500000,17.922865,\Rx:=0.000000,\Ry:=0.600766),vel1,zoneval,Extruder\WObj:=Workobject_1;
MoveL RelTool (p1,43.000000,11.500000,17.994972,\Rx:=0.000000,\Ry:=0.006657),vel1,zoneval,Extruder\WObj:=Workobject_1;
MoveL RelTool (p1,40.500000,11.500000,17.933304,\Rx:=0.000000,\Ry:=-0.765887),vel1,zoneval,Extruder\WObj:=Workobject_1;
MoveL RelTool (p1,38.000000,11.500000,17.727216,\Rx:=0.000000,\Ry:=-1.345493),vel1,zoneval,Extruder\WObj:=Workobject_1;
MoveL RelTool (p1,35.500000,11.500000,17.389298,\Rx:=0.000000,\Ry:=-2.131683),vel1,zoneval,Extruder\WObj:=Workobject_1;
MoveL RelTool (p1,33.000000,11.500000,16.882120,\Rx:=0.000000,\Ry:=-2.914944),vel1,zoneval,Extruder\WObj:=Workobject_1;
MoveL RelTool (p1,30.500000,11.500000,16.221969,\Rx:=0.000000,\Ry:=-4.017459),vel1,zoneval,Extruder\WObj:=Workobject_1;
MoveL RelTool (p1,28.000000,11.500000,15.346011,\Rx:=0.000000,\Ry:=-5.184167),vel1,zoneval,Extruder\WObj:=Workobject_1;
MoveL RelTool (p1,25.500000,11.500000,14.204898,\Rx:=0.000000,\Ry:=-6.237915),vel1,zoneval,Extruder\WObj:=Workobject_1;
MoveL RelTool (p1,23.000000,11.500000,12.681723,\Rx:=0.000000,\Ry:=-8.103445),vel1,zoneval,Extruder\WObj:=Workobject_1;
MoveL RelTool (p1,20.500000,11.500000,10.429283,\Rx:=0.000000,\Ry:=-11.215567),vel1,zoneval,Extruder\WObj:=Workobject_1;
MoveL RelTool (p1,18.000000,11.500000,8.180767,\Rx:=0.000000,\Ry:=-3.082616),vel1,zoneval,Extruder\WObj:=Workobject_1;
MoveL RelTool (p1,15.500000,11.500000,8.000000,\Rx:=0.000000,\Ry:=0.000000),vel1,zoneval,Extruder\WObj:=Workobject_1;
MoveL RelTool (p1,13.000000,11.500000,8.000000,\Rx:=0.000000,\Ry:=0.000000),vel1,zoneval,Extruder\WObj:=Workobject_1;
MoveL RelTool (p1,10.500000,11.500000,8.000000,\Rx:=0.000000,\Ry:=0.000000),vel1,zoneval,Extruder\WObj:=Workobject_1;
MoveL RelTool (p1,8.000000,11.500000,8.000000,\Rx:=0.000000,\Ry:=0.000000),vel1,zoneval,Extruder\WObj:=Workobject_1;
MoveL RelTool (p1,5.500000,11.500000,8.000000,\Rx:=0.000000,\Ry:=0.000000),vel1,zoneval,Extruder\WObj:=Workobject_1;
MoveL RelTool (p1,3.000000,11.500000,8.000000,\Rx:=0.000000,\Ry:=0.000000),vel1,zoneval,Extruder\WObj:=Workobject_1;
MoveL RelTool (p1,5.000000,12.000000,8.000000,\Rx:=0.000000,\Ry:=-0.000000),vel1,zoneval,Extruder\WObj:=Workobject_1;
MoveL RelTool (p1,7.500000,12.000000,8.000000,\Rx:=0.000000,\Ry:=-0.000000),vel1,zoneval,Extruder\WObj:=Workobject_1;
MoveL RelTool (p1,10.000000,12.000000,8.000000,\Rx:=0.000000,\Ry:=-0.000000),vel1,zoneval,Extruder\WObj:=Workobject_1;
MoveL RelTool (p1,12.500000,12.000000,8.000000,\Rx:=0.000000,\Ry:=-0.000000),vel1,zoneval,Extruder\WObj:=Workobject_1;
MoveL RelTool (p1,15.000000,12.000000,8.000000,\Rx:=0.000000,\Ry:=-0.000000),vel1,zoneval,Extruder\WObj:=Workobject_1;
MoveL RelTool (p1,17.500000,12.000000,8.057291,\Rx:=0.000000,\Ry:=-3.082616),vel1,zoneval,Extruder\WObj:=Workobject_1;
MoveL RelTool (p1,20.000000,12.000000,9.823128,\Rx:=0.000000,\Ry:=-11.222919),vel1,zoneval,Extruder\WObj:=Workobject_1;
MoveL RelTool (p1,22.500000,12.000000,12.313046,\Rx:=0.000000,\Ry:=-8.083750),vel1,zoneval,Extruder\WObj:=Workobject_1;
